(* CoDeSys 2.3.4.1 project: 20191210SRL乘3.pro *)
(* Libraries: Hollysys_PLC_COMM.lib 5.3.08 09:34:58, Hollysys_PLC_ANALOG.lib 28.12.05 14:28:34, Util.lib 28.10.11 18:19:34, SysLibVisu.lib 28.12.05 14:28:34, Hollysys_PLC_AnalogConvert.lib 5.3.08 09:47:22, Hollysys_PLC_Math.lib 7.3.06 16:53:32, Standard.lib 6.12.05 17:07:52, Hollysys_PLC_COMM2.lib 5.3.08 09:34:50, SYSLIBCALLBACK.LIB 6.12.05 17:07:52, Hollysys_PLC_Ex.lib 28.12.05 14:28:28, HS_PLC_ModebusMaster.lib 26.7.11 11:59:52 *)

(* PLC configuration (modules and I/O channels)
I AT %ID0 [DWORDInput_bit] 24 channels digital input
Q AT %QW0 [WordOutput3108_bit] 16 channels digital output(Relay)
LM3222 8×DO Relay [Ext_DO8_RELAY] node 0, in %IB4 out %QB2
  AT %QW2 [WordOutput_bit] 8 channels digital output(Relay)
LM3231 4×DI 4×DO Relay [Ext_DI4_DO4_RELAY] node 1, in %IB4 out %QB4
  AT %QW4 [WordOutput_bit] 4 channels digital output(Relay)
  AT %IW4 [WordInput_bit] 4 channels digital input
*)

(* POU PLC_PRG, LD *)
 PROGRAM PLC_PRG
VAR

	PSH_Q: BOOL;
	PSH_BL: BLINK;
	ET: TIME;
	KJ_SUO: BOOL;
	DY_SUO: BOOL;
	TD_TON: TON;
	TD_TON_Q: BOOL;
	PSH_BL_YSJ: BLINK;
	PSH_Q_YSJ: BOOL;
	JQ_1: JIQI_KONGZHI;
	JQ_2: JIQI_KONGZHI;
	JQ_JSH: ZJSHQ;
	CHD_1: BOOL;
	CHD_4: BOOL;
	CHD_3: BOOL;
	CHD_2: BOOL;
	BH_JQ_1: BAOHU_XIANSHI;
	YSJ_ONE_50_1: BOOL;
	YSJ_ONE_75_1: BOOL;
	YSJ_ONE_100_1: BOOL;
	YSJ_TWO_50_1: BOOL;
	YSJ_TWO_75_1: BOOL;
	YSJ_TWO_100_1: BOOL;
	T_DIAN: BOOL;
	T_R: R_TRIG;
	BH_JQ_2: BAOHU_XIANSHI;
	LN_SHB: BH_ZHFL;
	YOUFEN: YOU_FEN;

	MM_SUO: SUO;
	LN_FSH_1: BH_ZHFL;

	CHT: BOOL := 1;
	PW_OUT AT %MW892: INT;
	LN_FSH_2: BH_ZHFL;
	JT_KA: BOOL;
	YALI_OUT_1 AT %MW882: INT;
	PQ_YL_OUT AT %MW884: INT;
	PQ_XZH AT %MW364: INT;
	FAN_1_KA: BOOL;
	FAN_2_KA: BOOL;
	SHB_KA: BOOL;
	YL_KA: BOOL;
	PQYL: PQ_ZHFL_KZH;
	JZ_NJ_SHU_1: WORD;
	XUZH_IN_1 AT %MW476: INT;
	HIGH_IN_1 AT %MW478: INT;
	LOW_IN_1 AT %MW480: INT;
	XH_YSH_1: XH_YANSHI_1;
	XH_NJ_1: JQ_NJ_SHU;


	JJQ_DCF_1: BOOL;
	JQ_BJ_1: BJ_MIN_COOL;
	JQ_FUWEI_1: BJ_FUWEI;
	JQ_XHPX_1: XH_PAIXU;
	A_CX_1: BYTE;
	B_CX_1: BYTE;
       C_CX_1: BYTE;
	D_CX_1: BYTE;
	E_CX_1: BYTE;
	FU_WEI_1: BOOL;
	YSJ_ONE_1: BOOL;
	YSJ_TWO_1: BOOL;
	WBKZH: BOOL;
	XQ_1_T AT %MW886: INT;
	GRD_1_OUT AT %MW890: WORD;
	GRD_1_YSH: WORD;






	YL_FAN: BH_ZHFL;
	KF_ALA: BOOL;




	YSJ_CHD: BOOL;
	DY_JT: DY_JT_KZH;
	DY_JT_ALA: BOOL;
	CHD_5: BOOL;
	CHD_6: BOOL;
	F_CX_1: BYTE;
	YSJ_ONE: BOOL;
	YSJ_ONE_50: BOOL;
	YSJ_ONE_75: BOOL;
	YSJ_ONE_100: BOOL;
	YSJ_TWO: BOOL;
	YSJ_TWO_50: BOOL;
	YSJ_TWO_75: BOOL;
	YSJ_TWO_100: BOOL;
	YSJ_THREE: BOOL;
	YSJ_THREE_50: BOOL;
	YSJ_THREE_75: BOOL;
	YSJ_THREE_100: BOOL;
	YSJ_FOUR: BOOL;
	YSJ_FOUR_50: BOOL;
	YSJ_FOUR_75: BOOL;
	YSJ_FOUR_100: BOOL;
	YSJ_FIVE: BOOL;
	YSJ_FIVE_50: BOOL;
	YSJ_FIVE_75: BOOL;
	YSJ_FIVE_100: BOOL;
	YSJ_SIX: BOOL;
	YSJ_SIX_50: BOOL;
	YSJ_SIX_75: BOOL;
	YSJ_SIX_100: BOOL;

	BH_JQ_3: BAOHU_XIANSHI;
	JQ_3: JIQI_KONGZHI;
	BH_JQ_4: BAOHU_XIANSHI;
	JQ_4: JIQI_KONGZHI;
	BH_JQ_5: BAOHU_XIANSHI;
	JQ_5: JIQI_KONGZHI;
	BH_JQ_6: BAOHU_XIANSHI;
	JQ_6: JIQI_KONGZHI;
	PW_MN: MONI_LIANG_PW;

	PT_P: BLINK;

	GGD: AN_NIU;

	FAN_3_KA: BOOL;
	SHB2_KA: BOOL;
	FAN1: BH_ZHFL;
	FAN2: BH_ZHFL;
	FAN3: BH_ZHFL;
	YL: BH_ZHFL;
	SHB2: BH_ZHFL;
	SHB: BH_ZHFL;


	XQ_WD_XZH AT %MW470: INT;
	BH_WD AT %MW888: INT;
	PQ_YA_OUT AT %MW884: INT;


	Set_Local_Address: Set_Local_Address;
	MOUDBAS_OUT: BOOL;

	Analog_O: BOOL;
	FAN_4_KA: BOOL;
	OPEN_KJ: OPEN_KJ;
	FAN4: BH_ZHFL;






	R1_WD AT %MW1012: INT;
	R2_WD AT %MW1022: INT;
	R3_WD AT %MW1032: INT;
	R4_WD AT %MW1042: INT;
	R5_WD AT %MW1052: INT;
	R6_WD AT %MW1062: INT;
	R7_WD AT %MW1072: INT;
	R8_WD AT %MW1082: INT;

	R9_WD AT %MW1092: INT;
	R10_WD AT %MW1102: INT;
	R11_WD AT %MW1112: INT;
	R12_WD AT %MW1122: INT;
	R13_WD AT %MW1132: INT;
	R14_WD AT %MW1142: INT;






	K1: AN_NIU;
	K2: AN_NIU;
	K3: AN_NIU;
	K4: AN_NIU;
	K5: AN_NIU;
	K6: AN_NIU;
	K7: AN_NIU;
	K8: AN_NIU;
	K9: AN_NIU;
	K10: AN_NIU;
	K11: AN_NIU;
	K12: AN_NIU;
	K13: AN_NIU;
	K14: AN_NIU;


	K1_XZ AT %MW610: INT;
	K2_XZ AT %MW620: INT;
	K3_XZ AT %MW630: INT;
	K4_XZ AT %MW640: INT;
	K5_XZ AT %MW650: INT;
	K6_XZ AT %MW660: INT;
	K7_XZ AT %MW670: INT;
	K8_XZ AT %MW680: INT;
	K9_XZ AT %MW690: INT;
	K10_XZ AT %MW500: INT;
	K11_XZ AT %MW510: INT;
	K12_XZ AT %MW520: INT;
	K13_XZ AT %MW530: INT;
	K14_XZ AT %MW540: INT;

	K1_KJ AT %MW612: INT;
	K2_KJ AT %MW622: INT;
	K3_KJ AT %MW632: INT;
	K4_KJ AT %MW642: INT;
	K5_KJ AT %MW652: INT;
	K6_KJ AT %MW662: INT;
	K7_KJ AT %MW672: INT;
	K8_KJ AT %MW682: INT;
	K9_KJ AT %MW692: INT;
	K10_KJ AT %MW502: INT;
	K11_KJ AT %MW512: INT;
	K12_KJ AT %MW522: INT;
	K13_KJ AT %MW532: INT;
	K14_KJ AT %MW542: INT;


	K1_TJ AT %MW614: INT;
	K2_TJ AT %MW624: INT;
	K3_TJ AT %MW634: INT;
	K4_TJ AT %MW644: INT;
	K5_TJ AT %MW654: INT;
	K6_TJ AT %MW664: INT;
	K7_TJ AT %MW674: INT;
	K8_TJ AT %MW684: INT;
	K9_TJ AT %MW694: INT;
	K10_TJ AT %MW504: INT;
	K11_TJ AT %MW514: INT;
	K12_TJ AT %MW524: INT;
	K13_TJ AT %MW534: INT;
	K14_TJ AT %MW544: INT;

	K1_GS AT %MW616: INT;
	K2_GS AT %MW626: INT;
	K3_GS AT %MW636: INT;
	K4_GS AT %MW646: INT;
	K5_GS AT %MW656: INT;
	K6_GS AT %MW666: INT;
	K7_GS AT %MW676: INT;
	K8_GS AT %MW686: INT;
	K9_GS AT %MW696: INT;
	K10_GS AT %MW506: INT;
	K11_GS AT %MW516: INT;
	K12_GS AT %MW526: INT;
	K13_GS AT %MW536: INT;
	K14_GS AT %MW546: INT;


	DEF_1: BOOL;
	DEF_2: BOOL;
	DEF_3: BOOL;
	DEF_4: BOOL;
	DEF_5: BOOL;
	DEF_6: BOOL;
	DEF_7: BOOL;
	DEF_8: BOOL;
	DEF_9: BOOL;
	DEF_10: BOOL;
	DEF_11: BOOL;
	DEF_12: BOOL;
	DEF_13: BOOL;
	DEF_14: BOOL;
	DEF_1_DD: BOOL;
	DEF_2_DD: BOOL;
	DEF_3_DD: BOOL;
	DEF_4_DD: BOOL;
	DEF_5_DD: BOOL;
	DEF_6_DD: BOOL;
	DEF_7_DD: BOOL;
	DEF_8_DD: BOOL;
	DEF_9_DD: BOOL;
	DEF_10_DD: BOOL;
	DEF_11_DD: BOOL;
	DEF_12_DD: BOOL;
	DEF_13_DD: BOOL;
	DEF_14_DD: BOOL;
	ROOM1_ALA: BOOL;
	ROOM2_ALA: BOOL;
	ROOM3_ALA: BOOL;
	ROOM4_ALA: BOOL;
	ROOM5_ALA: BOOL;
	ROOM6_ALA: BOOL;
	ROOM7_ALA: BOOL;
	ROOM8_ALA: BOOL;
	ROOM9_ALA: BOOL;
	ROOM10_ALA: BOOL;
	ROOM11_ALA: BOOL;
	ROOM12_ALA: BOOL;
	ROOM13_ALA: BOOL;
	ROOM14_ALA: BOOL;
	COOL_1_M: DWORD;
	COOL_2_M: DWORD;
	COOL_3_M: DWORD;
	COOL_4_M: DWORD;
	COOL_5_M: DWORD;
	COOL_6_M: DWORD;
	COOL_7_M: DWORD;
	COOL_8_M: DWORD;
	COOL_9_M: DWORD;
	COOL_10_M: DWORD;
	COOL_11_M: DWORD;
	COOL_12_M: DWORD;
	COOL_13_M: DWORD;
	COOL_14_M: DWORD;
	ROOM1_T_ZT: WORD;
	ROOM2_T_ZT: WORD;
	ROOM3_T_ZT: WORD;
	ROOM4_T_ZT: WORD;
	ROOM5_T_ZT: WORD;
	ROOM6_T_ZT: WORD;
	ROOM7_T_ZT: WORD;
	ROOM8_T_ZT: WORD;
	ROOM9_T_ZT: WORD;
	ROOM10_T_ZT: WORD;
	ROOM11_T_ZT: WORD;
	ROOM12_T_ZT: WORD;
	ROOM13_T_ZT: WORD;
	ROOM14_T_ZT: WORD;
	BZH_1_M: DWORD;
	BZH_2_M: DWORD;
	BZH_3_M: DWORD;
	BZH_4_M: DWORD;
	BZH_5_M: DWORD;
	BZH_6_M: DWORD;
	BZH_7_M: DWORD;
	BZH_8_M: DWORD;
	BZH_9_M: DWORD;
	BZH_10_M: DWORD;
	BZH_11_M: DWORD;
	BZH_12_M: DWORD;
	BZH_13_M: DWORD;
	BZH_14_M: DWORD;

	DEF_1_ZD: BOOL;
	DEF_2_ZD: BOOL;
	DEF_3_ZD: BOOL;
	DEF_4_ZD: BOOL;
	DEF_5_ZD: BOOL;
	DEF_6_ZD: BOOL;
	DEF_7_ZD: BOOL;
	DEF_8_ZD: BOOL;
	DEF_9_ZD: BOOL;
	DEF_10_ZD: BOOL;
	DEF_11_ZD: BOOL;
	DEF_12_ZD: BOOL;
	DEF_13_ZD: BOOL;
	DEF_14_ZD: BOOL;

	DEF_1_FJ: BOOL;
	DEF_2_FJ: BOOL;
	DEF_3_FJ: BOOL;
	DEF_4_FJ: BOOL;
	DEF_5_FJ: BOOL;
	DEF_6_FJ: BOOL;
	DEF_7_FJ: BOOL;
	DEF_8_FJ: BOOL;
	DEF_9_FJ: BOOL;
	DEF_10_FJ: BOOL;
	DEF_11_FJ: BOOL;
	DEF_12_FJ: BOOL;
	DEF_13_FJ: BOOL;
	DEF_14_FJ: BOOL;

	ROOM_1_FJ: BOOL;
	ROOM_2_FJ: BOOL;
	ROOM_3_FJ: BOOL;
	ROOM_4_FJ: BOOL;
	ROOM_5_FJ: BOOL;
	ROOM_6_FJ: BOOL;
	ROOM_7_FJ: BOOL;
	ROOM_8_FJ: BOOL;
	ROOM_9_FJ: BOOL;
	ROOM_10_FJ: BOOL;
	ROOM_11_FJ: BOOL;
	ROOM_12_FJ: BOOL;
	ROOM_13_FJ: BOOL;
	ROOM_14_FJ: BOOL;



	DEF_YUNSUAN: DEF_YUNSUAN;

	CS_SHB: BH_ZHFL;
	YL_K: BH_ZHFL;

	CF: BLINK;

	Analog_: BOOL;
	OPEN_K: OPEN_KJ;
	Analog_IN1: Analog_IN;
	Analog_OUT1: BOOL;
	Analog_IN2: Analog_IN;
	Analog_OUT2: BOOL;

	FB1_CHD: BOOL;
	FB1_ALA: BOOL;
	FB2_CHD: BOOL;
	FB2_ALA: BOOL;

	FB_AN: AN_NIU;
	FB_TON: TON;
	YW_XSH AT %MW1200: INT;
	SS: BOOL;


	B1: BOOL;
	B3: BOOL;
	B2: BOOL;
	XZ_NIU: AN_NIU;
	BY_NIU: AN_NIU;
	FB_CHD: BOOL;
	WBKZH1: BOOL;
	PQ_GRD: PQ_GRD;
	PQ_BH_WD AT %MW906: INT;
	PQ_GRD_OUT AT %MW908: INT;
	PQ_GRD_SET AT %MW490: INT;
	HQ_WD_XZ AT %MW598: INT;
	KCHD_1: BOOL;
	KCHD_2: BOOL;
	KCHD_3: BOOL;
	KCHD_4: BOOL;
	DEF_SHB: BH_ZHFL;

	Analog_IN3: Analog_IN;
	Analog_OUT3: BOOL;

	TT_BH_WCH AT %MW448: INT;
	SHB_YAN: YANSHI_CLOSE;
	SHL_YSH_SET AT %MW468: WORD;
	SHL_YSH_SET_0: BOOL;
	SHL_T: YANSHI_OPEN;
	SHL_BH: SHL_BH;
	KJ: BOOL;
	SHB1: BOOL;

	T1 AT %MW1300: INT;
	T2 AT %MW1302: INT;
	JQ_BJ: BJ_MIN_COOL_1;
	JQ_FUWEI: BJ_FUWEI_1;
	FW_1: BOOL;
	FW_3: BOOL;
	FW_2: BOOL;
	FW_4: BOOL;
	FW_5: BOOL;
	FW_6: BOOL;
	CX_1: BYTE;
	CX_2: BYTE;
	CX_3: BYTE;
	CX_4: BYTE;
	CX_5: BYTE;
	CX_6: BYTE;




	WD_XH1: WD_XH;
	K1_IN: INT;
	K1_T1 AT %MW1300: INT;
	K1_T2 AT %MW1302: INT;
	K1_T3 AT %MW1304: INT;
	K1_T4 AT %MW1306: INT;

	K2_T1 AT %MW1308: INT;
	K2_T2 AT %MW1310: INT;
	K2_T3 AT %MW1312: INT;
	K2_T4 AT %MW1314: INT;

	K3_T1 AT %MW1316: INT;
	K3_T2 AT %MW1318: INT;

	K3_T4 AT %MW1322: INT;
	K4_T1 AT %MW1324: INT;
	K4_T2 AT %MW1326: INT;
	K4_T3 AT %MW1328: INT;
	K4_T4 AT %MW1330: INT;

	K2_IN: INT;
	WD_XH2: WD_XH;
	WD_XH3: WD_XH;
	K3_IN: INT;
	WD_XH4: WD_XH;
	K4_IN: INT;

	K3_T3 AT %MW1320: INT;
	Reset_COMM2_PRMT: Reset_COMM2_PRMT;
	Reset_COMM2_: BOOL;
	BLINK: BLINK;
	ModbusMaster485: ModbusMaster485;
	DDD: BYTE;
	ModbusMaster: BOOL;
	H: BOOL;
	O: BOOL;
	KCHD_5: BOOL;
	JQ_SHU: WORD;
	YL_DCF2: BOOL;
	TON_GYW: TON;
	SHB_AN: AN_NIU;
	BLINK_SHB: BLINK;
	SHB_XHKA: BOOL;
	YF_WD AT %MW1332: INT;
	K_1: BOOL;
	K_2: BOOL;
	YA_ALA: BOOL;
	YA AT %MW1332: INT;
	YA_CHA AT %MW1334: INT;
	SET_YA AT %MW618: INT;
	Y_K: BOOL;
	JJQ: BOOL;
	JJQ_K AT %MW628: INT;
	JJQ_G AT %MW638: INT;
	BB: BB;
	HIGH_IN_2 AT %MW648: INT;
	LOW_IN_2 AT %MW658: INT;
END_VAR
VAR RETAIN

END_VAR
VAR RETAIN
END_VAR
VAR_INPUT
END_VAR
VAR_OUTPUT
END_VAR
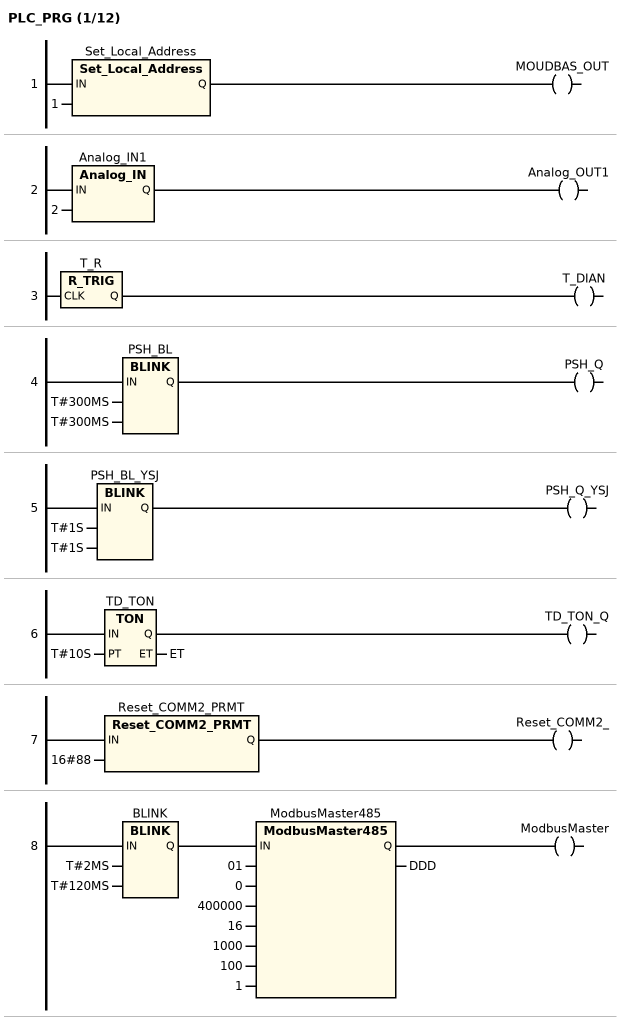
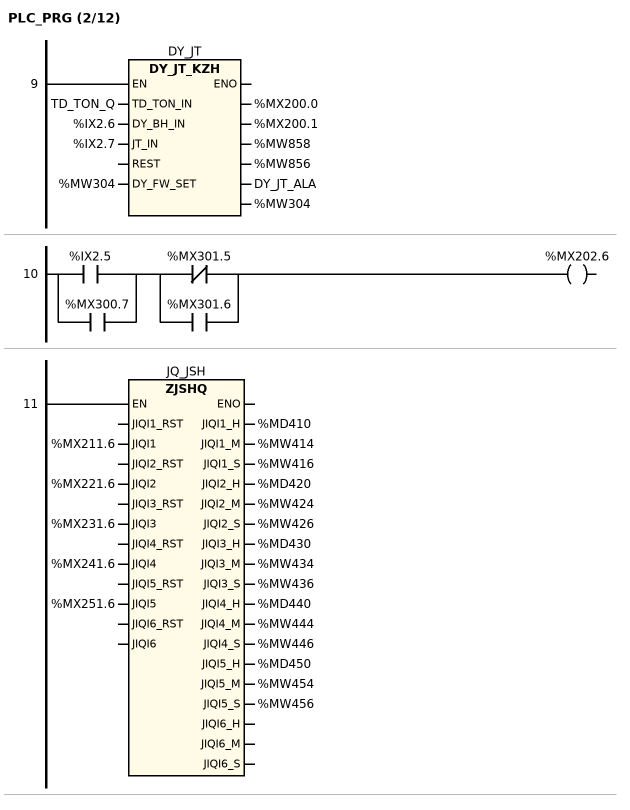
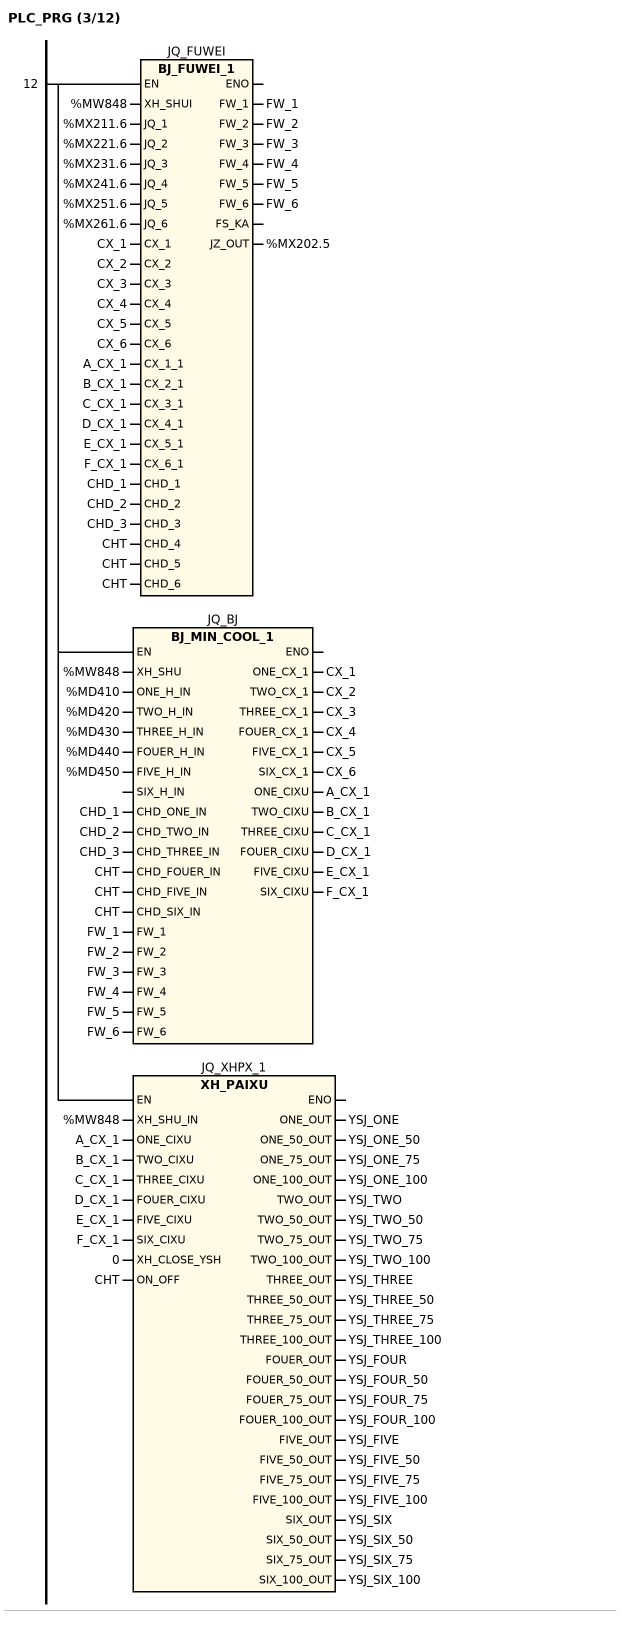
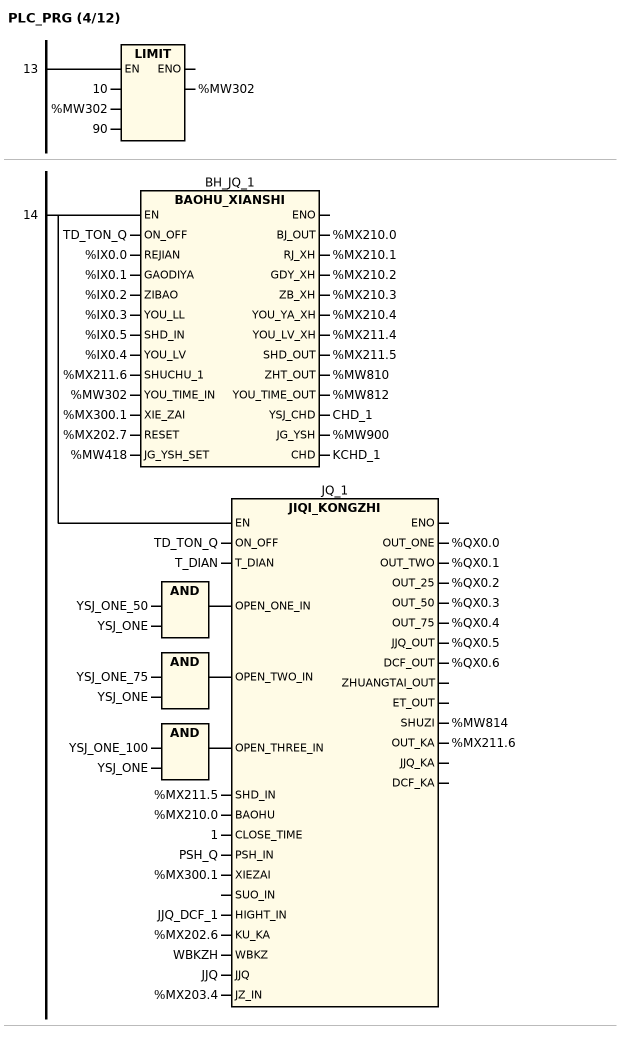
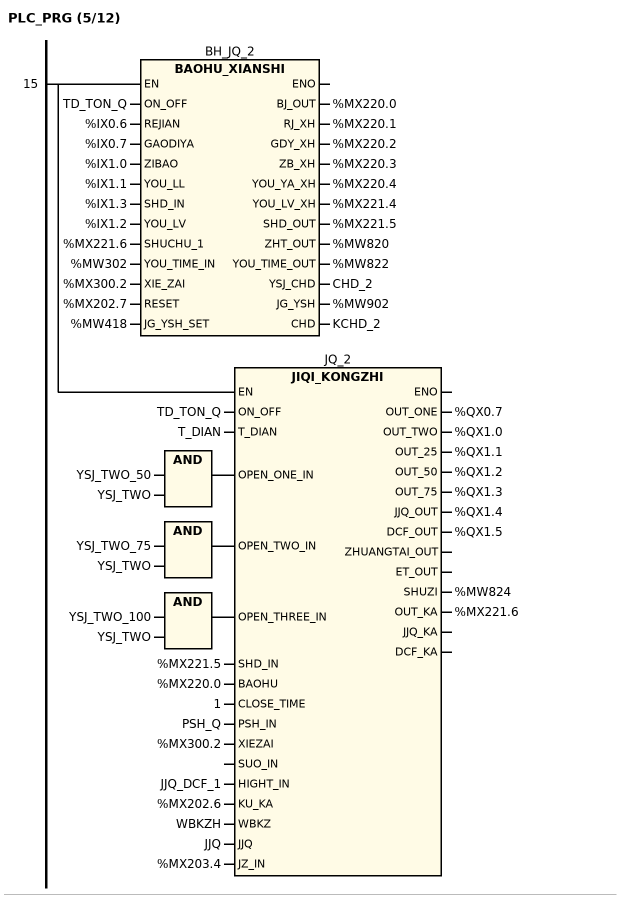
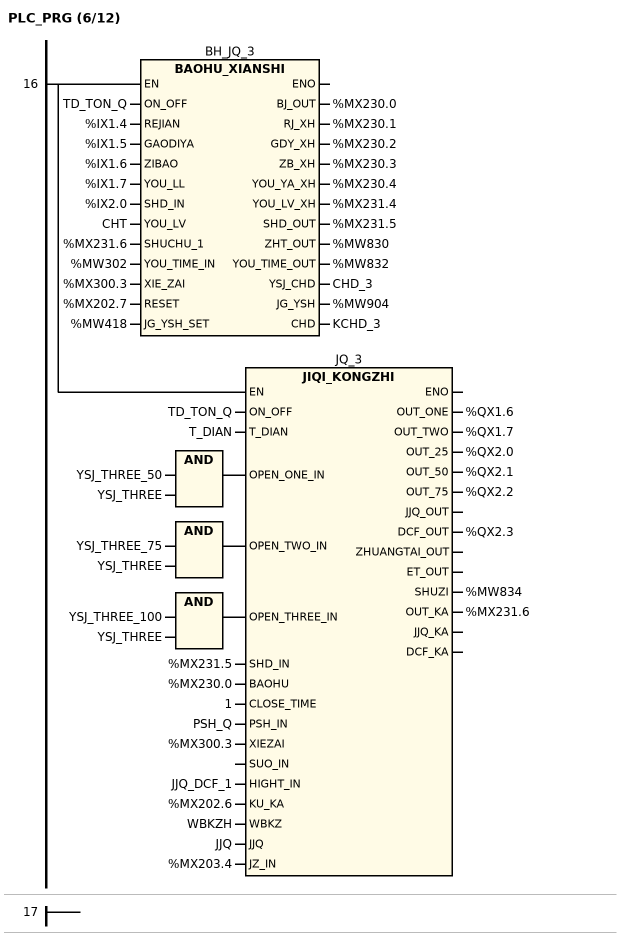
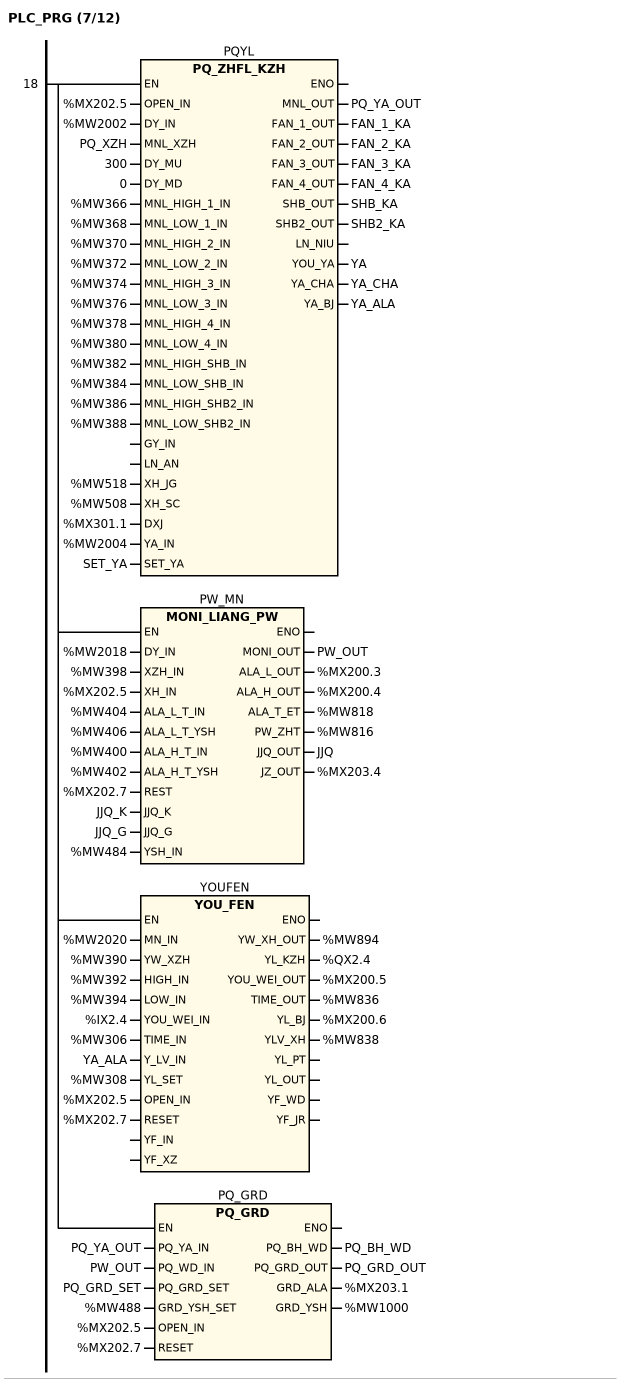
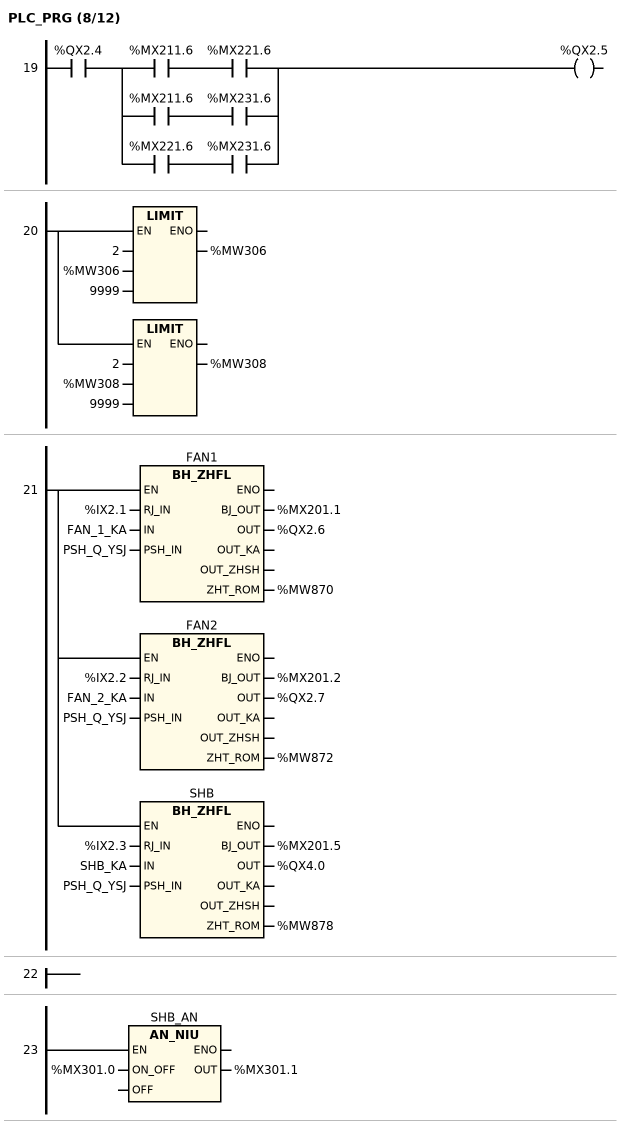
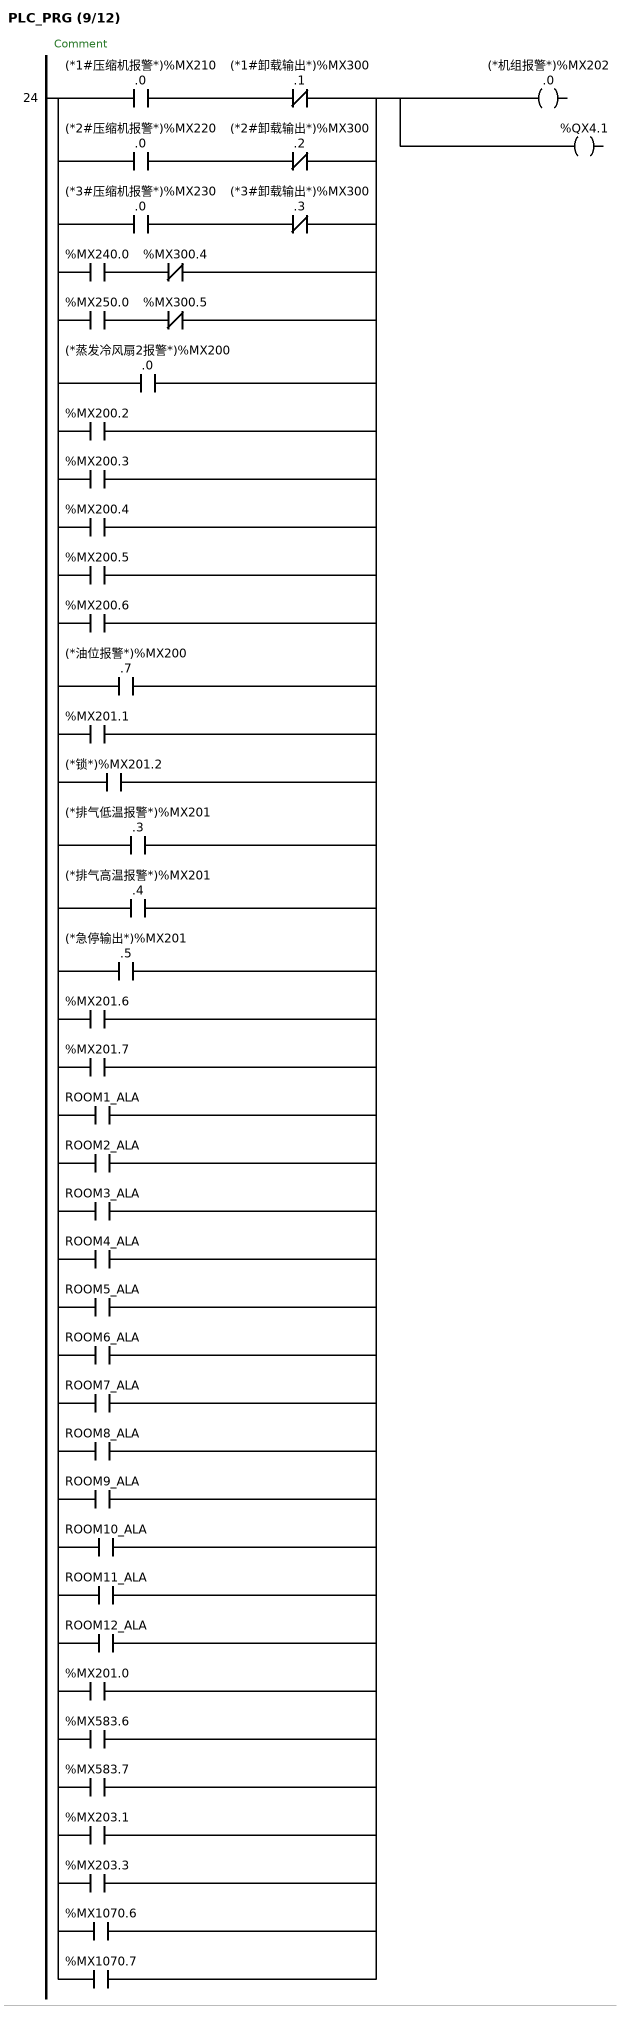
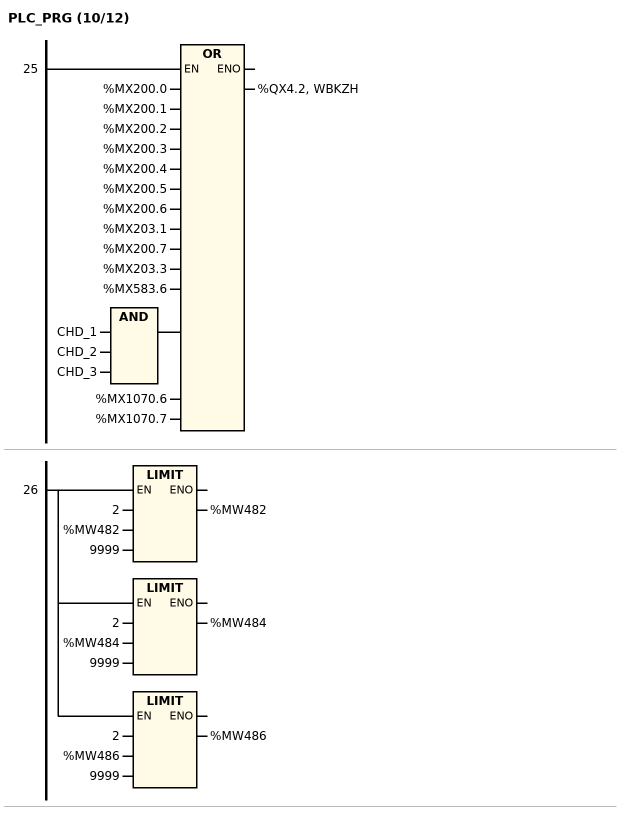
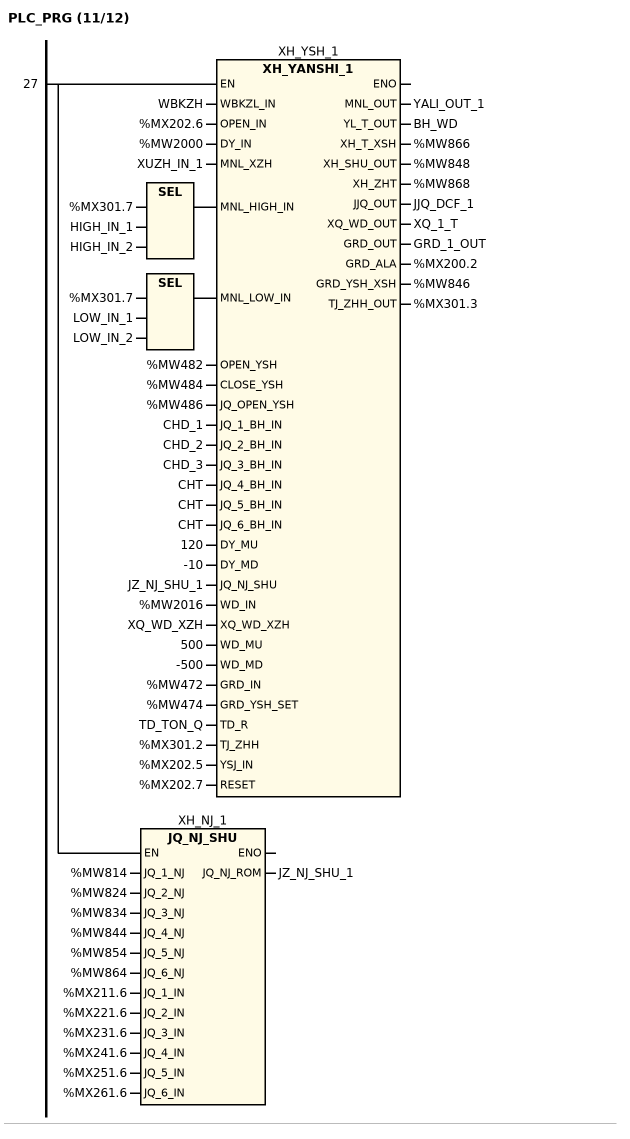
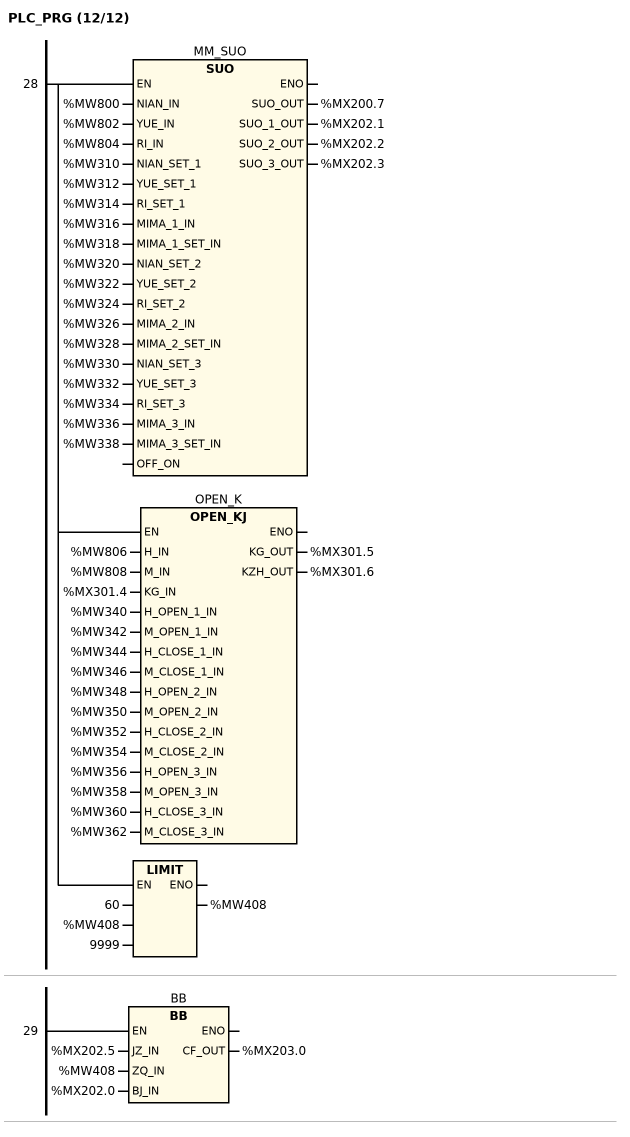
_LD_ (* Ladder Diagram *)
NETWORK 1
	Set_Local_Address:Set_Local_Address(*, 1) --- (MOUDBAS_OUT)
NETWORK 2
	Analog_IN1:Analog_IN(*, 2) --- (Analog_OUT1)
NETWORK 3
	T_R:R_TRIG(CLK: *) --- (T_DIAN)
NETWORK 4
	PSH_BL:BLINK(*, T#300MS, T#300MS) --- (PSH_Q)
NETWORK 5
	PSH_BL_YSJ:BLINK(*, T#1S, T#1S) --- (PSH_Q_YSJ)
NETWORK 6
	TD_TON:TON(IN: *, PT: T#10S, ET => ET) --- (TD_TON_Q)
NETWORK 7
	Reset_COMM2_PRMT:Reset_COMM2_PRMT(*, 16#88) --- (Reset_COMM2_)
NETWORK 8
	BLINK:BLINK(*, T#2MS, T#120MS) - ModbusMaster485:ModbusMaster485(*, 01, 0, 400000, 16, 1000, 100, 1, out 2 => DDD) --- (ModbusMaster)
NETWORK 9
	*
		EN --- DY_JT:DY_JT_KZH(TD_TON_IN: TD_TON_Q, DY_BH_IN: %IX2.6, JT_IN: %IX2.7, REST: , DY_FW_SET: %MW304, out 2 => %MX200.1, out 3 => %MW858, out 4 => %MW856, out 5 => DY_JT_ALA, out 6 => %MW304) => %MX200.0
NETWORK 10
	{ [%IX2.5] | [%MX300.7] } - { [/%MX301.5] | [%MX301.6] } --- (%MX202.6)
NETWORK 11
	*
		EN --- JQ_JSH:ZJSHQ(JIQI1_RST: , JIQI1: %MX211.6, JIQI2_RST: , JIQI2: %MX221.6, JIQI3_RST: , JIQI3: %MX231.6, JIQI4_RST: , JIQI4: %MX241.6, JIQI5_RST: , JIQI5: %MX251.6, JIQI6_RST: , JIQI6: , JIQI1_M => %MW414, JIQI1_S => %MW416, JIQI2_H => %MD420, JIQI2_M => %MW424, JIQI2_S => %MW426, JIQI3_H => %MD430, JIQI3_M => %MW434, JIQI3_S => %MW436, JIQI4_H => %MD440, JIQI4_M => %MW444, JIQI4_S => %MW446, JIQI5_H => %MD450, JIQI5_M => %MW454, JIQI5_S => %MW456) => %MD410
NETWORK 12
	*
		EN --- JQ_FUWEI:BJ_FUWEI_1(XH_SHUI: %MW848, JQ_1: %MX211.6, JQ_2: %MX221.6, JQ_3: %MX231.6, JQ_4: %MX241.6, JQ_5: %MX251.6, JQ_6: %MX261.6, CX_1: CX_1, CX_2: CX_2, CX_3: CX_3, CX_4: CX_4, CX_5: CX_5, CX_6: CX_6, CX_1_1: A_CX_1, CX_2_1: B_CX_1, CX_3_1: C_CX_1, CX_4_1: D_CX_1, CX_5_1: E_CX_1, CX_6_1: F_CX_1, CHD_1: CHD_1, CHD_2: CHD_2, CHD_3: CHD_3, CHD_4: CHT, CHD_5: CHT, CHD_6: CHT, FW_2 => FW_2, FW_3 => FW_3, FW_4 => FW_4, FW_5 => FW_5, FW_6 => FW_6, JZ_OUT => %MX202.5) => FW_1
		EN --- JQ_BJ:BJ_MIN_COOL_1(XH_SHU: %MW848, ONE_H_IN: %MD410, TWO_H_IN: %MD420, THREE_H_IN: %MD430, FOUER_H_IN: %MD440, FIVE_H_IN: %MD450, SIX_H_IN: , CHD_ONE_IN: CHD_1, CHD_TWO_IN: CHD_2, CHD_THREE_IN: CHD_3, CHD_FOUER_IN: CHT, CHD_FIVE_IN: CHT, CHD_SIX_IN: CHT, FW_1: FW_1, FW_2: FW_2, FW_3: FW_3, FW_4: FW_4, FW_5: FW_5, FW_6: FW_6, TWO_CX_1 => CX_2, THREE_CX_1 => CX_3, FOUER_CX_1 => CX_4, FIVE_CX_1 => CX_5, SIX_CX_1 => CX_6, ONE_CIXU => A_CX_1, TWO_CIXU => B_CX_1, THREE_CIXU => C_CX_1, FOUER_CIXU => D_CX_1, FIVE_CIXU => E_CX_1, SIX_CIXU => F_CX_1) => CX_1
		EN --- JQ_XHPX_1:XH_PAIXU(XH_SHU_IN: %MW848, ONE_CIXU: A_CX_1, TWO_CIXU: B_CX_1, THREE_CIXU: C_CX_1, FOUER_CIXU: D_CX_1, FIVE_CIXU: E_CX_1, SIX_CIXU: F_CX_1, XH_CLOSE_YSH: 0, ON_OFF: CHT, ONE_50_OUT => YSJ_ONE_50, ONE_75_OUT => YSJ_ONE_75, ONE_100_OUT => YSJ_ONE_100, TWO_OUT => YSJ_TWO, TWO_50_OUT => YSJ_TWO_50, TWO_75_OUT => YSJ_TWO_75, TWO_100_OUT => YSJ_TWO_100, THREE_OUT => YSJ_THREE, THREE_50_OUT => YSJ_THREE_50, THREE_75_OUT => YSJ_THREE_75, THREE_100_OUT => YSJ_THREE_100, FOUER_OUT => YSJ_FOUR, FOUER_50_OUT => YSJ_FOUR_50, FOUER_75_OUT => YSJ_FOUR_75, FOUER_100_OUT => YSJ_FOUR_100, FIVE_OUT => YSJ_FIVE, FIVE_50_OUT => YSJ_FIVE_50, FIVE_75_OUT => YSJ_FIVE_75, FIVE_100_OUT => YSJ_FIVE_100, SIX_OUT => YSJ_SIX, SIX_50_OUT => YSJ_SIX_50, SIX_75_OUT => YSJ_SIX_75, SIX_100_OUT => YSJ_SIX_100) => YSJ_ONE
NETWORK 13
	*
		EN --- LIMIT(10, %MW302, 90) => %MW302
NETWORK 14
	*
		EN --- BH_JQ_1:BAOHU_XIANSHI(ON_OFF: TD_TON_Q, REJIAN: %IX0.0, GAODIYA: %IX0.1, ZIBAO: %IX0.2, YOU_LL: %IX0.3, SHD_IN: %IX0.5, YOU_LV: %IX0.4, SHUCHU_1: %MX211.6, YOU_TIME_IN: %MW302, XIE_ZAI: %MX300.1, RESET: %MX202.7, JG_YSH_SET: %MW418, RJ_XH => %MX210.1, GDY_XH => %MX210.2, ZB_XH => %MX210.3, YOU_YA_XH => %MX210.4, YOU_LV_XH => %MX211.4, SHD_OUT => %MX211.5, ZHT_OUT => %MW810, YOU_TIME_OUT => %MW812, YSJ_CHD => CHD_1, JG_YSH => %MW900, CHD => KCHD_1) => %MX210.0
		EN --- JQ_1:JIQI_KONGZHI(ON_OFF: TD_TON_Q, T_DIAN: T_DIAN, OPEN_ONE_IN: AND(YSJ_ONE_50, YSJ_ONE), OPEN_TWO_IN: AND(YSJ_ONE_75, YSJ_ONE), OPEN_THREE_IN: AND(YSJ_ONE_100, YSJ_ONE), SHD_IN: %MX211.5, BAOHU: %MX210.0, CLOSE_TIME: 1, PSH_IN: PSH_Q, XIEZAI: %MX300.1, SUO_IN: , HIGHT_IN: JJQ_DCF_1, KU_KA: %MX202.6, WBKZ: WBKZH, JJQ: JJQ, JZ_IN: %MX203.4, OUT_TWO => %QX0.1, OUT_25 => %QX0.2, OUT_50 => %QX0.3, OUT_75 => %QX0.4, JJQ_OUT => %QX0.5, DCF_OUT => %QX0.6, SHUZI => %MW814, OUT_KA => %MX211.6) => %QX0.0
NETWORK 15
	*
		EN --- BH_JQ_2:BAOHU_XIANSHI(ON_OFF: TD_TON_Q, REJIAN: %IX0.6, GAODIYA: %IX0.7, ZIBAO: %IX1.0, YOU_LL: %IX1.1, SHD_IN: %IX1.3, YOU_LV: %IX1.2, SHUCHU_1: %MX221.6, YOU_TIME_IN: %MW302, XIE_ZAI: %MX300.2, RESET: %MX202.7, JG_YSH_SET: %MW418, RJ_XH => %MX220.1, GDY_XH => %MX220.2, ZB_XH => %MX220.3, YOU_YA_XH => %MX220.4, YOU_LV_XH => %MX221.4, SHD_OUT => %MX221.5, ZHT_OUT => %MW820, YOU_TIME_OUT => %MW822, YSJ_CHD => CHD_2, JG_YSH => %MW902, CHD => KCHD_2) => %MX220.0
		EN --- JQ_2:JIQI_KONGZHI(ON_OFF: TD_TON_Q, T_DIAN: T_DIAN, OPEN_ONE_IN: AND(YSJ_TWO_50, YSJ_TWO), OPEN_TWO_IN: AND(YSJ_TWO_75, YSJ_TWO), OPEN_THREE_IN: AND(YSJ_TWO_100, YSJ_TWO), SHD_IN: %MX221.5, BAOHU: %MX220.0, CLOSE_TIME: 1, PSH_IN: PSH_Q, XIEZAI: %MX300.2, SUO_IN: , HIGHT_IN: JJQ_DCF_1, KU_KA: %MX202.6, WBKZ: WBKZH, JJQ: JJQ, JZ_IN: %MX203.4, OUT_TWO => %QX1.0, OUT_25 => %QX1.1, OUT_50 => %QX1.2, OUT_75 => %QX1.3, JJQ_OUT => %QX1.4, DCF_OUT => %QX1.5, SHUZI => %MW824, OUT_KA => %MX221.6) => %QX0.7
NETWORK 16
	*
		EN --- BH_JQ_3:BAOHU_XIANSHI(ON_OFF: TD_TON_Q, REJIAN: %IX1.4, GAODIYA: %IX1.5, ZIBAO: %IX1.6, YOU_LL: %IX1.7, SHD_IN: %IX2.0, YOU_LV: CHT, SHUCHU_1: %MX231.6, YOU_TIME_IN: %MW302, XIE_ZAI: %MX300.3, RESET: %MX202.7, JG_YSH_SET: %MW418, RJ_XH => %MX230.1, GDY_XH => %MX230.2, ZB_XH => %MX230.3, YOU_YA_XH => %MX230.4, YOU_LV_XH => %MX231.4, SHD_OUT => %MX231.5, ZHT_OUT => %MW830, YOU_TIME_OUT => %MW832, YSJ_CHD => CHD_3, JG_YSH => %MW904, CHD => KCHD_3) => %MX230.0
		EN --- JQ_3:JIQI_KONGZHI(ON_OFF: TD_TON_Q, T_DIAN: T_DIAN, OPEN_ONE_IN: AND(YSJ_THREE_50, YSJ_THREE), OPEN_TWO_IN: AND(YSJ_THREE_75, YSJ_THREE), OPEN_THREE_IN: AND(YSJ_THREE_100, YSJ_THREE), SHD_IN: %MX231.5, BAOHU: %MX230.0, CLOSE_TIME: 1, PSH_IN: PSH_Q, XIEZAI: %MX300.3, SUO_IN: , HIGHT_IN: JJQ_DCF_1, KU_KA: %MX202.6, WBKZ: WBKZH, JJQ: JJQ, JZ_IN: %MX203.4, OUT_TWO => %QX1.7, OUT_25 => %QX2.0, OUT_50 => %QX2.1, OUT_75 => %QX2.2, DCF_OUT => %QX2.3, SHUZI => %MW834, OUT_KA => %MX231.6) => %QX1.6
NETWORK 17
	*
NETWORK 18
	*
		EN --- PQYL:PQ_ZHFL_KZH(OPEN_IN: %MX202.5, DY_IN: %MW2002, MNL_XZH: PQ_XZH, DY_MU: 300, DY_MD: 0, MNL_HIGH_1_IN: %MW366, MNL_LOW_1_IN: %MW368, MNL_HIGH_2_IN: %MW370, MNL_LOW_2_IN: %MW372, MNL_HIGH_3_IN: %MW374, MNL_LOW_3_IN: %MW376, MNL_HIGH_4_IN: %MW378, MNL_LOW_4_IN: %MW380, MNL_HIGH_SHB_IN: %MW382, MNL_LOW_SHB_IN: %MW384, MNL_HIGH_SHB2_IN: %MW386, MNL_LOW_SHB2_IN: %MW388, GY_IN: , LN_AN: , XH_JG: %MW518, XH_SC: %MW508, DXJ: %MX301.1, YA_IN: %MW2004, SET_YA: SET_YA, FAN_1_OUT => FAN_1_KA, FAN_2_OUT => FAN_2_KA, FAN_3_OUT => FAN_3_KA, FAN_4_OUT => FAN_4_KA, SHB_OUT => SHB_KA, SHB2_OUT => SHB2_KA, YOU_YA => YA, YA_CHA => YA_CHA, YA_BJ => YA_ALA) => PQ_YA_OUT
		EN --- PW_MN:MONI_LIANG_PW(DY_IN: %MW2018, XZH_IN: %MW398, XH_IN: %MX202.5, ALA_L_T_IN: %MW404, ALA_L_T_YSH: %MW406, ALA_H_T_IN: %MW400, ALA_H_T_YSH: %MW402, REST: %MX202.7, JJQ_K: JJQ_K, JJQ_G: JJQ_G, YSH_IN: %MW484, ALA_L_OUT => %MX200.3, ALA_H_OUT => %MX200.4, ALA_T_ET => %MW818, PW_ZHT => %MW816, JJQ_OUT => JJQ, JZ_OUT => %MX203.4) => PW_OUT
		EN --- YOUFEN:YOU_FEN(MN_IN: %MW2020, YW_XZH: %MW390, HIGH_IN: %MW392, LOW_IN: %MW394, YOU_WEI_IN: %IX2.4, TIME_IN: %MW306, Y_LV_IN: YA_ALA, YL_SET: %MW308, OPEN_IN: %MX202.5, RESET: %MX202.7, YF_IN: , YF_XZ: , YL_KZH => %QX2.4, YOU_WEI_OUT => %MX200.5, TIME_OUT => %MW836, YL_BJ => %MX200.6, YLV_XH => %MW838) => %MW894
		EN --- PQ_GRD:PQ_GRD(PQ_YA_IN: PQ_YA_OUT, PQ_WD_IN: PW_OUT, PQ_GRD_SET: PQ_GRD_SET, GRD_YSH_SET: %MW488, OPEN_IN: %MX202.5, RESET: %MX202.7, PQ_GRD_OUT => PQ_GRD_OUT, GRD_ALA => %MX203.1, GRD_YSH => %MW1000) => PQ_BH_WD
NETWORK 19
	[%QX2.4] - { [%MX211.6] - [%MX221.6] | [%MX211.6] - [%MX231.6] | [%MX221.6] - [%MX231.6] } --- (%QX2.5)
NETWORK 20
	*
		EN --- LIMIT(2, %MW306, 9999) => %MW306
		EN --- LIMIT(2, %MW308, 9999) => %MW308
NETWORK 21
	*
		EN --- FAN1:BH_ZHFL(RJ_IN: %IX2.1, IN: FAN_1_KA, PSH_IN: PSH_Q_YSJ, OUT => %QX2.6, ZHT_ROM => %MW870) => %MX201.1
		EN --- FAN2:BH_ZHFL(RJ_IN: %IX2.2, IN: FAN_2_KA, PSH_IN: PSH_Q_YSJ, OUT => %QX2.7, ZHT_ROM => %MW872) => %MX201.2
		EN --- SHB:BH_ZHFL(RJ_IN: %IX2.3, IN: SHB_KA, PSH_IN: PSH_Q_YSJ, OUT => %QX4.0, ZHT_ROM => %MW878) => %MX201.5
NETWORK 22
	*
NETWORK 23
	*
		EN --- SHB_AN:AN_NIU(ON_OFF: %MX301.0, OFF: ) => %MX301.1
NETWORK 24 (* Comment *)
	{ [(*1#压缩机报警*)%MX210.0] - [/(*1#卸载输出*)%MX300.1] | [(*2#压缩机报警*)%MX220.0] - [/(*2#卸载输出*)%MX300.2] | [(*3#压缩机报警*)%MX230.0] - [/(*3#卸载输出*)%MX300.3] | [%MX240.0] - [/%MX300.4] | [%MX250.0] - [/%MX300.5] | [(*蒸发冷风扇2报警*)%MX200.0] | [%MX200.2] | [%MX200.3] | [%MX200.4] | [%MX200.5] | [%MX200.6] | [(*油位报警*)%MX200.7] | [%MX201.1] | [(*锁*)%MX201.2] | [(*排气低温报警*)%MX201.3] | [(*排气高温报警*)%MX201.4] | [(*急停输出*)%MX201.5] | [%MX201.6] | [%MX201.7] | [ROOM1_ALA] | [ROOM2_ALA] | [ROOM3_ALA] | [ROOM4_ALA] | [ROOM5_ALA] | [ROOM6_ALA] | [ROOM7_ALA] | [ROOM8_ALA] | [ROOM9_ALA] | [ROOM10_ALA] | [ROOM11_ALA] | [ROOM12_ALA] | [%MX201.0] | [%MX583.6] | [%MX583.7] | [%MX203.1] | [%MX203.3] | [%MX1070.6] | [%MX1070.7] } --- ((*机组报警*)%MX202.0) (%QX4.1)
NETWORK 25
	*
		EN --- OR(%MX200.0, %MX200.1, %MX200.2, %MX200.3, %MX200.4, %MX200.5, %MX200.6, %MX203.1, %MX200.7, %MX203.3, %MX583.6, AND(CHD_1, CHD_2, CHD_3), %MX1070.6, %MX1070.7) => %QX4.2, WBKZH
NETWORK 26
	*
		EN --- LIMIT(2, %MW482, 9999) => %MW482
		EN --- LIMIT(2, %MW484, 9999) => %MW484
		EN --- LIMIT(2, %MW486, 9999) => %MW486
NETWORK 27
	*
		EN --- XH_YSH_1:XH_YANSHI_1(WBKZL_IN: WBKZH, OPEN_IN: %MX202.6, DY_IN: %MW2000, MNL_XZH: XUZH_IN_1, MNL_HIGH_IN: SEL(%MX301.7, HIGH_IN_1, HIGH_IN_2), MNL_LOW_IN: SEL(%MX301.7, LOW_IN_1, LOW_IN_2), OPEN_YSH: %MW482, CLOSE_YSH: %MW484, JQ_OPEN_YSH: %MW486, JQ_1_BH_IN: CHD_1, JQ_2_BH_IN: CHD_2, JQ_3_BH_IN: CHD_3, JQ_4_BH_IN: CHT, JQ_5_BH_IN: CHT, JQ_6_BH_IN: CHT, DY_MU: 120, DY_MD: -10, JQ_NJ_SHU: JZ_NJ_SHU_1, WD_IN: %MW2016, XQ_WD_XZH: XQ_WD_XZH, WD_MU: 500, WD_MD: -500, GRD_IN: %MW472, GRD_YSH_SET: %MW474, TD_R: TD_TON_Q, TJ_ZHH: %MX301.2, YSJ_IN: %MX202.5, RESET: %MX202.7, YL_T_OUT => BH_WD, XH_T_XSH => %MW866, XH_SHU_OUT => %MW848, XH_ZHT => %MW868, JJQ_OUT => JJQ_DCF_1, XQ_WD_OUT => XQ_1_T, GRD_OUT => GRD_1_OUT, GRD_ALA => %MX200.2, GRD_YSH_XSH => %MW846, TJ_ZHH_OUT => %MX301.3) => YALI_OUT_1
		EN --- XH_NJ_1:JQ_NJ_SHU(JQ_1_NJ: %MW814, JQ_2_NJ: %MW824, JQ_3_NJ: %MW834, JQ_4_NJ: %MW844, JQ_5_NJ: %MW854, JQ_6_NJ: %MW864, JQ_1_IN: %MX211.6, JQ_2_IN: %MX221.6, JQ_3_IN: %MX231.6, JQ_4_IN: %MX241.6, JQ_5_IN: %MX251.6, JQ_6_IN: %MX261.6) => JZ_NJ_SHU_1
NETWORK 28
	*
		EN --- MM_SUO:SUO(NIAN_IN: %MW800, YUE_IN: %MW802, RI_IN: %MW804, NIAN_SET_1: %MW310, YUE_SET_1: %MW312, RI_SET_1: %MW314, MIMA_1_IN: %MW316, MIMA_1_SET_IN: %MW318, NIAN_SET_2: %MW320, YUE_SET_2: %MW322, RI_SET_2: %MW324, MIMA_2_IN: %MW326, MIMA_2_SET_IN: %MW328, NIAN_SET_3: %MW330, YUE_SET_3: %MW332, RI_SET_3: %MW334, MIMA_3_IN: %MW336, MIMA_3_SET_IN: %MW338, OFF_ON: , SUO_1_OUT => %MX202.1, SUO_2_OUT => %MX202.2, SUO_3_OUT => %MX202.3) => %MX200.7
		EN --- OPEN_K:OPEN_KJ(H_IN: %MW806, M_IN: %MW808, KG_IN: %MX301.4, H_OPEN_1_IN: %MW340, M_OPEN_1_IN: %MW342, H_CLOSE_1_IN: %MW344, M_CLOSE_1_IN: %MW346, H_OPEN_2_IN: %MW348, M_OPEN_2_IN: %MW350, H_CLOSE_2_IN: %MW352, M_CLOSE_2_IN: %MW354, H_OPEN_3_IN: %MW356, M_OPEN_3_IN: %MW358, H_CLOSE_3_IN: %MW360, M_CLOSE_3_IN: %MW362, KZH_OUT => %MX301.6) => %MX301.5
		EN --- LIMIT(60, %MW408, 9999) => %MW408
NETWORK 29
	*
		EN --- BB:BB(JZ_IN: %MX202.5, ZQ_IN: %MW408, BJ_IN: %MX202.0) => %MX203.0
_END_LD_
(* the same logic as Structured Text *)
(* Network 1: see the listing above *)
(* Network 2: see the listing above *)
(* Network 3 *)
T_R(CLK := TRUE);
T_DIAN := T_R.Q;
(* Network 4: see the listing above *)
(* Network 5: see the listing above *)
(* Network 6 *)
TD_TON(IN := TRUE, PT := T#10S);
ET := TD_TON.ET;
TD_TON_Q := TD_TON.Q;
(* Network 7: see the listing above *)
(* Network 8: see the listing above *)
(* Network 9: see the listing above *)
(* Network 10 *)
%MX202.6 := (%IX2.5 OR %MX300.7) AND (NOT %MX301.5 OR %MX301.6);
(* Network 11: see the listing above *)
(* Network 12: see the listing above *)
(* Network 13 *)
%MW302 := LIMIT(10, %MW302, 90);
(* Network 14: see the listing above *)
(* Network 15: see the listing above *)
(* Network 16: see the listing above *)
(* Network 17: see the listing above *)
(* Network 18: see the listing above *)
(* Network 19 *)
%QX2.5 := %QX2.4 AND (%MX211.6 AND %MX221.6 OR %MX211.6 AND %MX231.6 OR %MX221.6 AND %MX231.6);
(* Network 20 *)
%MW306 := LIMIT(2, %MW306, 9999);
%MW308 := LIMIT(2, %MW308, 9999);
(* Network 21 *)
FAN1(RJ_IN := %IX2.1, IN := FAN_1_KA, PSH_IN := PSH_Q_YSJ);
%QX2.6 := FAN1.OUT;
%MW870 := FAN1.ZHT_ROM;
%MX201.1 := FAN1.BJ_OUT;
FAN2(RJ_IN := %IX2.2, IN := FAN_2_KA, PSH_IN := PSH_Q_YSJ);
%QX2.7 := FAN2.OUT;
%MW872 := FAN2.ZHT_ROM;
%MX201.2 := FAN2.BJ_OUT;
SHB(RJ_IN := %IX2.3, IN := SHB_KA, PSH_IN := PSH_Q_YSJ);
%QX4.0 := SHB.OUT;
%MW878 := SHB.ZHT_ROM;
%MX201.5 := SHB.BJ_OUT;
(* Network 22: see the listing above *)
(* Network 23: see the listing above *)
(* Network 24 *)
(*机组报警*)%MX202.0 := ((*1#压缩机报警*)%MX210.0) AND NOT ((*1#卸载输出*)%MX300.1) OR ((*2#压缩机报警*)%MX220.0) AND NOT ((*2#卸载输出*)%MX300.2) OR ((*3#压缩机报警*)%MX230.0) AND NOT ((*3#卸载输出*)%MX300.3) OR %MX240.0 AND NOT %MX300.4 OR %MX250.0 AND NOT %MX300.5 OR ((*蒸发冷风扇2报警*)%MX200.0) OR %MX200.2 OR %MX200.3 OR %MX200.4 OR %MX200.5 OR %MX200.6 OR ((*油位报警*)%MX200.7) OR %MX201.1 OR ((*锁*)%MX201.2) OR ((*排气低温报警*)%MX201.3) OR ((*排气高温报警*)%MX201.4) OR ((*急停输出*)%MX201.5) OR %MX201.6 OR %MX201.7 OR ROOM1_ALA OR ROOM2_ALA OR ROOM3_ALA OR ROOM4_ALA OR ROOM5_ALA OR ROOM6_ALA OR ROOM7_ALA OR ROOM8_ALA OR ROOM9_ALA OR ROOM10_ALA OR ROOM11_ALA OR ROOM12_ALA OR %MX201.0 OR %MX583.6 OR %MX583.7 OR %MX203.1 OR %MX203.3 OR %MX1070.6 OR %MX1070.7;
%QX4.1 := (*机组报警*)%MX202.0;
(* Network 25: see the listing above *)
(* Network 26 *)
%MW482 := LIMIT(2, %MW482, 9999);
%MW484 := LIMIT(2, %MW484, 9999);
%MW486 := LIMIT(2, %MW486, 9999);
(* Network 27 *)
XH_YSH_1(WBKZL_IN := WBKZH, OPEN_IN := %MX202.6, DY_IN := %MW2000, MNL_XZH := XUZH_IN_1, MNL_HIGH_IN := SEL(%MX301.7, HIGH_IN_1, HIGH_IN_2), MNL_LOW_IN := SEL(%MX301.7, LOW_IN_1, LOW_IN_2), OPEN_YSH := %MW482, CLOSE_YSH := %MW484, JQ_OPEN_YSH := %MW486, JQ_1_BH_IN := CHD_1, JQ_2_BH_IN := CHD_2, JQ_3_BH_IN := CHD_3, JQ_4_BH_IN := CHT, JQ_5_BH_IN := CHT, JQ_6_BH_IN := CHT, DY_MU := 120, DY_MD := -10, JQ_NJ_SHU := JZ_NJ_SHU_1, WD_IN := %MW2016, XQ_WD_XZH := XQ_WD_XZH, WD_MU := 500, WD_MD := -500, GRD_IN := %MW472, GRD_YSH_SET := %MW474, TD_R := TD_TON_Q, TJ_ZHH := %MX301.2, YSJ_IN := %MX202.5, RESET := %MX202.7);
BH_WD := XH_YSH_1.YL_T_OUT;
%MW866 := XH_YSH_1.XH_T_XSH;
%MW848 := XH_YSH_1.XH_SHU_OUT;
%MW868 := XH_YSH_1.XH_ZHT;
JJQ_DCF_1 := XH_YSH_1.JJQ_OUT;
XQ_1_T := XH_YSH_1.XQ_WD_OUT;
GRD_1_OUT := XH_YSH_1.GRD_OUT;
%MX200.2 := XH_YSH_1.GRD_ALA;
%MW846 := XH_YSH_1.GRD_YSH_XSH;
%MX301.3 := XH_YSH_1.TJ_ZHH_OUT;
YALI_OUT_1 := XH_YSH_1.MNL_OUT;
XH_NJ_1(JQ_1_NJ := %MW814, JQ_2_NJ := %MW824, JQ_3_NJ := %MW834, JQ_4_NJ := %MW844, JQ_5_NJ := %MW854, JQ_6_NJ := %MW864, JQ_1_IN := %MX211.6, JQ_2_IN := %MX221.6, JQ_3_IN := %MX231.6, JQ_4_IN := %MX241.6, JQ_5_IN := %MX251.6, JQ_6_IN := %MX261.6);
JZ_NJ_SHU_1 := XH_NJ_1.JQ_NJ_ROM;
(* Network 28: see the listing above *)
(* Network 29 *)
BB(JZ_IN := %MX202.5, ZQ_IN := %MW408, BJ_IN := %MX202.0);
%MX203.0 := BB.CF_OUT;
END_PROGRAM

(* POU JIQI_KONGZHI, LD *)
  FUNCTION_BLOCK JIQI_KONGZHI
VAR_INPUT
	ON_OFF: BOOL;
	T_DIAN: BOOL;
	OPEN_ONE_IN: BOOL;
	OPEN_TWO_IN: BOOL;
	OPEN_THREE_IN: BOOL;
	SHD_IN: BOOL;
       BAOHU: BOOL;
	CLOSE_TIME: WORD;
	PSH_IN: BOOL;
	XIEZAI: BOOL;
	SUO_IN: BOOL;
	HIGHT_IN: BOOL;
	KU_KA: BOOL;
	WBKZ: BOOL;
	JJQ: BOOL;
	JZ_IN: BOOL;
END_VAR
VAR_OUTPUT
	OUT_ONE: BOOL;
	OUT_TWO: BOOL;
	OUT_25: BOOL;
	OUT_50: BOOL;
	OUT_75: BOOL;
	JJQ_OUT: BOOL;
	DCF_OUT: BOOL;
	ZHUANGTAI_OUT: BOOL;
	ET_OUT: WORD;
	SHUZI: WORD;
	OUT_KA: BOOL;
	JJQ_KA: BOOL;
	DCF_KA: BOOL;
END_VAR
VAR
	T_YASHI: TON;
	BAOJING_OUT: BOOL;
	OUT_100: BOOL;
	ET_TON_YASHI: TIME;
	T_YASHI_Q: BOOL;
	CLOSE: YANSHI_CLOSE;
	TOF_25: TOF;
	ET_TOF_25: TIME;
	T_25: TON;
	ET_T_25: TIME;
	T_50: TON;
	ET_T_50: TIME;
	T_75: TON;
	ET_T_75: TIME;
	OUT_50_KA: BOOL;
	OUT_75_KA: BOOL;
	SHD_KA: BOOL;
	BLINK: BLINK;
	KA_OFF: BOOL;
	R_TRIG: R_TRIG;
	JSHU: WORD;
	R_QL: R_TRIG;
END_VAR
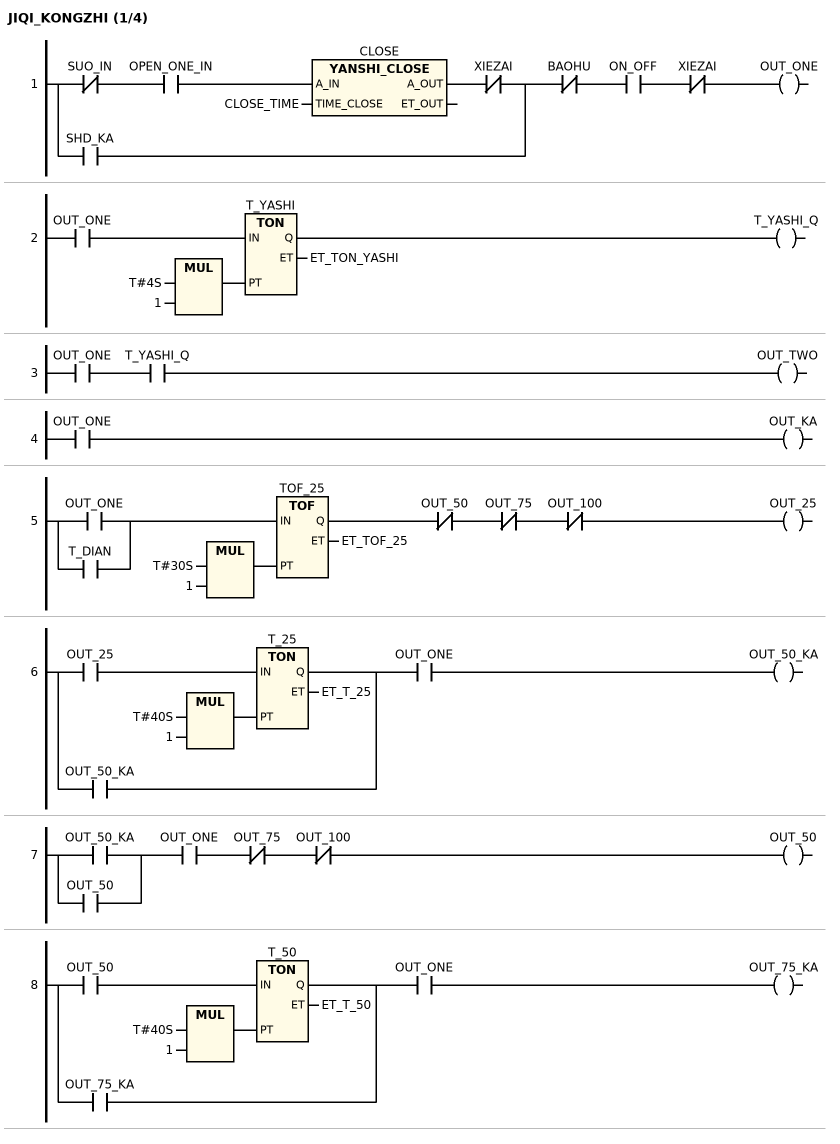
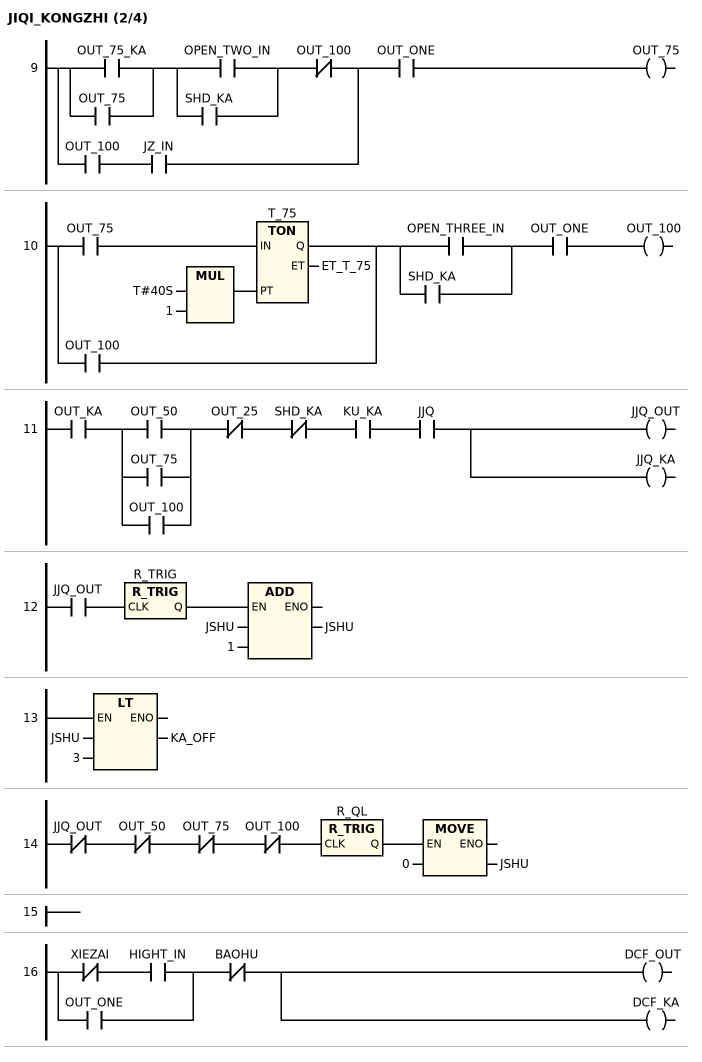
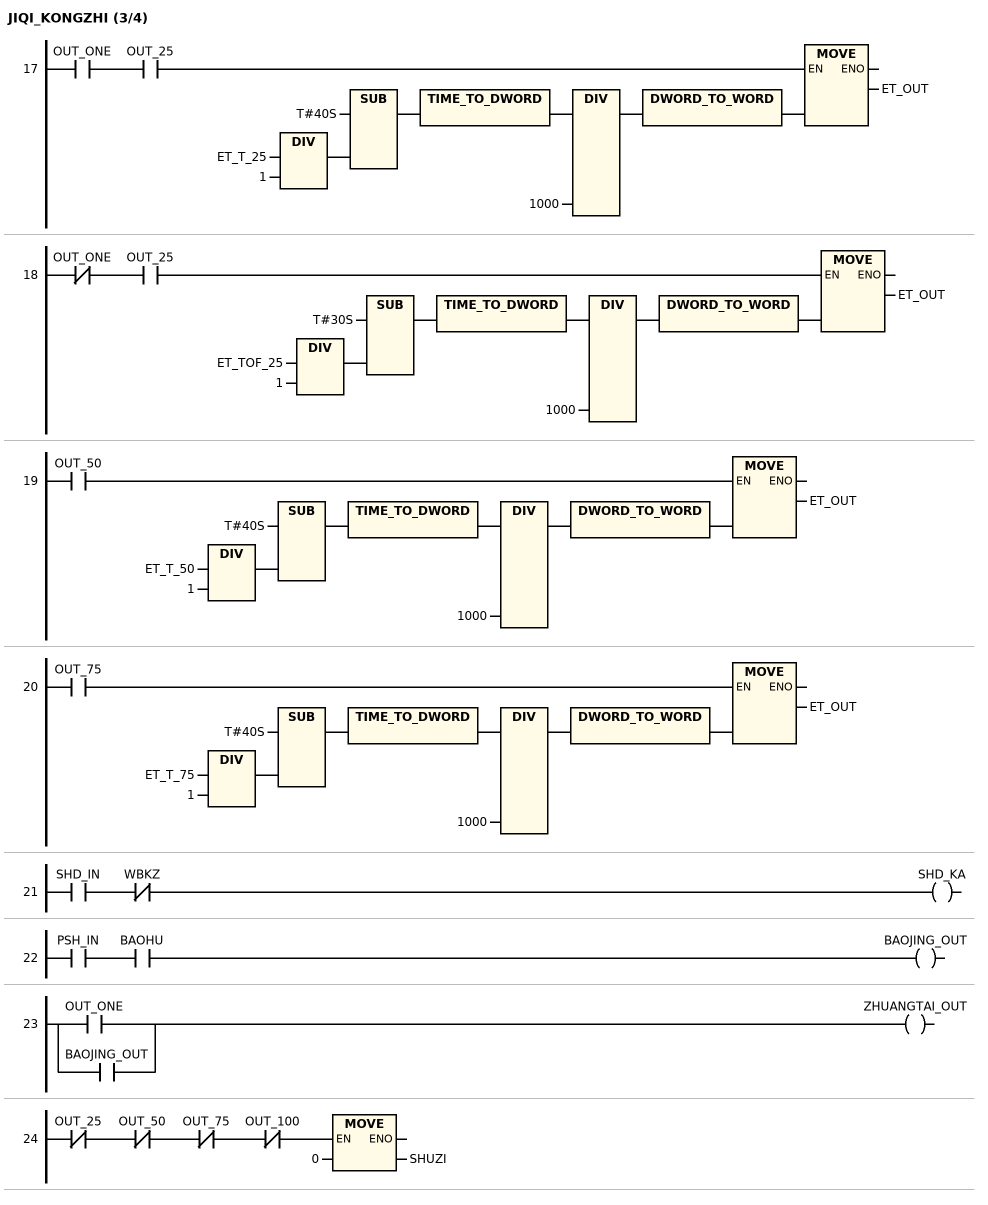
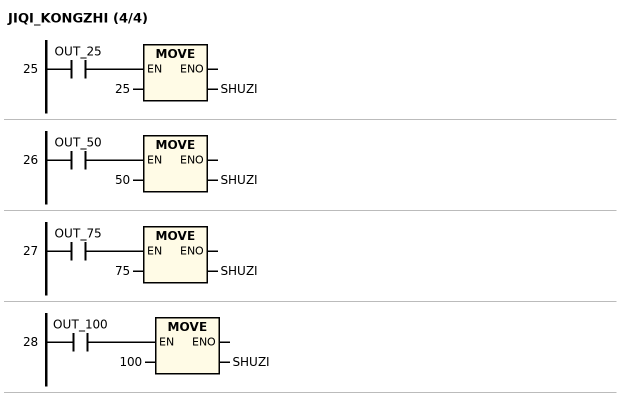
_LD_ (* Ladder Diagram *)
NETWORK 1
	{ [/SUO_IN] - [OPEN_ONE_IN] - CLOSE:YANSHI_CLOSE(A_IN: *, TIME_CLOSE: CLOSE_TIME) - [/XIEZAI] | [SHD_KA] } - [/BAOHU] - [ON_OFF] - [/XIEZAI] --- (OUT_ONE)
NETWORK 2
	[OUT_ONE] - T_YASHI:TON(IN: *, PT: MUL(T#4S, 1), ET => ET_TON_YASHI) --- (T_YASHI_Q)
NETWORK 3
	[OUT_ONE] - [T_YASHI_Q] --- (OUT_TWO)
NETWORK 4
	[OUT_ONE] --- (OUT_KA)
NETWORK 5
	{ [OUT_ONE] | [T_DIAN] } - TOF_25:TOF(IN: *, PT: MUL(T#30S, 1), ET => ET_TOF_25) - [/OUT_50] - [/OUT_75] - [/OUT_100] --- (OUT_25)
NETWORK 6
	{ [OUT_25] - T_25:TON(IN: *, PT: MUL(T#40S, 1), ET => ET_T_25) | [OUT_50_KA] } - [OUT_ONE] --- (OUT_50_KA)
NETWORK 7
	{ [OUT_50_KA] | [OUT_50] } - [OUT_ONE] - [/OUT_75] - [/OUT_100] --- (OUT_50)
NETWORK 8
	{ [OUT_50] - T_50:TON(IN: *, PT: MUL(T#40S, 1), ET => ET_T_50) | [OUT_75_KA] } - [OUT_ONE] --- (OUT_75_KA)
NETWORK 9
	{ { [OUT_75_KA] | [OUT_75] } - { [OPEN_TWO_IN] | [SHD_KA] } - [/OUT_100] | [OUT_100] - [JZ_IN] } - [OUT_ONE] --- (OUT_75)
NETWORK 10
	{ [OUT_75] - T_75:TON(IN: *, PT: MUL(T#40S, 1), ET => ET_T_75) | [OUT_100] } - { [OPEN_THREE_IN] | [SHD_KA] } - [OUT_ONE] --- (OUT_100)
NETWORK 11
	[OUT_KA] - { [OUT_50] | [OUT_75] | [OUT_100] } - [/OUT_25] - [/SHD_KA] - [KU_KA] - [JJQ] --- (JJQ_OUT) (JJQ_KA)
NETWORK 12
	[JJQ_OUT] - R_TRIG:R_TRIG(CLK: *)
		EN --- ADD(JSHU, 1) => JSHU
NETWORK 13
	*
		EN --- LT(JSHU, 3) => KA_OFF
NETWORK 14
	[/JJQ_OUT] - [/OUT_50] - [/OUT_75] - [/OUT_100] - R_QL:R_TRIG(CLK: *)
		EN --- MOVE(0) => JSHU
NETWORK 15
	*
NETWORK 16
	{ [/XIEZAI] - [HIGHT_IN] | [OUT_ONE] } - [/BAOHU] --- (DCF_OUT) (DCF_KA)
NETWORK 17
	[OUT_ONE] - [OUT_25]
		EN --- MOVE(DWORD_TO_WORD(DIV(TIME_TO_DWORD(SUB(T#40S, DIV(ET_T_25, 1))), 1000))) => ET_OUT
NETWORK 18
	[/OUT_ONE] - [OUT_25]
		EN --- MOVE(DWORD_TO_WORD(DIV(TIME_TO_DWORD(SUB(T#30S, DIV(ET_TOF_25, 1))), 1000))) => ET_OUT
NETWORK 19
	[OUT_50]
		EN --- MOVE(DWORD_TO_WORD(DIV(TIME_TO_DWORD(SUB(T#40S, DIV(ET_T_50, 1))), 1000))) => ET_OUT
NETWORK 20
	[OUT_75]
		EN --- MOVE(DWORD_TO_WORD(DIV(TIME_TO_DWORD(SUB(T#40S, DIV(ET_T_75, 1))), 1000))) => ET_OUT
NETWORK 21
	[SHD_IN] - [/WBKZ] --- (SHD_KA)
NETWORK 22
	[PSH_IN] - [BAOHU] --- (BAOJING_OUT)
NETWORK 23
	{ [OUT_ONE] | [BAOJING_OUT] } --- (ZHUANGTAI_OUT)
NETWORK 24
	[/OUT_25] - [/OUT_50] - [/OUT_75] - [/OUT_100]
		EN --- MOVE(0) => SHUZI
NETWORK 25
	[OUT_25]
		EN --- MOVE(25) => SHUZI
NETWORK 26
	[OUT_50]
		EN --- MOVE(50) => SHUZI
NETWORK 27
	[OUT_75]
		EN --- MOVE(75) => SHUZI
NETWORK 28
	[OUT_100]
		EN --- MOVE(100) => SHUZI
_END_LD_
(* the same logic as Structured Text *)
(* Network 1 *)
CLOSE(A_IN := NOT SUO_IN AND OPEN_ONE_IN, TIME_CLOSE := CLOSE_TIME);
OUT_ONE := (CLOSE.A_OUT AND NOT XIEZAI OR SHD_KA) AND NOT BAOHU AND ON_OFF AND NOT XIEZAI;
(* Network 2 *)
T_YASHI(IN := OUT_ONE, PT := T#4S * 1);
ET_TON_YASHI := T_YASHI.ET;
T_YASHI_Q := T_YASHI.Q;
(* Network 3 *)
OUT_TWO := OUT_ONE AND T_YASHI_Q;
(* Network 4 *)
OUT_KA := OUT_ONE;
(* Network 5 *)
TOF_25(IN := OUT_ONE OR T_DIAN, PT := T#30S * 1);
ET_TOF_25 := TOF_25.ET;
OUT_25 := TOF_25.Q AND NOT OUT_50 AND NOT OUT_75 AND NOT OUT_100;
(* Network 6 *)
T_25(IN := OUT_25, PT := T#40S * 1);
ET_T_25 := T_25.ET;
OUT_50_KA := (T_25.Q OR OUT_50_KA) AND OUT_ONE;
(* Network 7 *)
OUT_50 := (OUT_50_KA OR OUT_50) AND OUT_ONE AND NOT OUT_75 AND NOT OUT_100;
(* Network 8 *)
T_50(IN := OUT_50, PT := T#40S * 1);
ET_T_50 := T_50.ET;
OUT_75_KA := (T_50.Q OR OUT_75_KA) AND OUT_ONE;
(* Network 9 *)
OUT_75 := ((OUT_75_KA OR OUT_75) AND (OPEN_TWO_IN OR SHD_KA) AND NOT OUT_100 OR OUT_100 AND JZ_IN) AND OUT_ONE;
(* Network 10 *)
T_75(IN := OUT_75, PT := T#40S * 1);
ET_T_75 := T_75.ET;
OUT_100 := (T_75.Q OR OUT_100) AND (OPEN_THREE_IN OR SHD_KA) AND OUT_ONE;
(* Network 11 *)
JJQ_OUT := OUT_KA AND (OUT_50 OR OUT_75 OR OUT_100) AND NOT OUT_25 AND NOT SHD_KA AND KU_KA AND JJQ;
JJQ_KA := JJQ_OUT;
(* Network 12 *)
R_TRIG(CLK := JJQ_OUT);
IF R_TRIG.Q THEN
	JSHU := JSHU + 1;
END_IF;
(* Network 13 *)
KA_OFF := JSHU < 3;
(* Network 14 *)
R_QL(CLK := NOT JJQ_OUT AND NOT OUT_50 AND NOT OUT_75 AND NOT OUT_100);
IF R_QL.Q THEN
	JSHU := 0;
END_IF;
(* Network 15 *)
(* Network 16 *)
DCF_OUT := (NOT XIEZAI AND HIGHT_IN OR OUT_ONE) AND NOT BAOHU;
DCF_KA := DCF_OUT;
(* Network 17 *)
IF OUT_ONE AND OUT_25 THEN
	ET_OUT := DWORD_TO_WORD(TIME_TO_DWORD(T#40S - (ET_T_25 / 1)) / 1000);
END_IF;
(* Network 18 *)
IF NOT OUT_ONE AND OUT_25 THEN
	ET_OUT := DWORD_TO_WORD(TIME_TO_DWORD(T#30S - (ET_TOF_25 / 1)) / 1000);
END_IF;
(* Network 19 *)
IF OUT_50 THEN
	ET_OUT := DWORD_TO_WORD(TIME_TO_DWORD(T#40S - (ET_T_50 / 1)) / 1000);
END_IF;
(* Network 20 *)
IF OUT_75 THEN
	ET_OUT := DWORD_TO_WORD(TIME_TO_DWORD(T#40S - (ET_T_75 / 1)) / 1000);
END_IF;
(* Network 21 *)
SHD_KA := SHD_IN AND NOT WBKZ;
(* Network 22 *)
BAOJING_OUT := PSH_IN AND BAOHU;
(* Network 23 *)
ZHUANGTAI_OUT := OUT_ONE OR BAOJING_OUT;
(* Network 24 *)
IF NOT OUT_25 AND NOT OUT_50 AND NOT OUT_75 AND NOT OUT_100 THEN
	SHUZI := 0;
END_IF;
(* Network 25 *)
IF OUT_25 THEN
	SHUZI := 25;
END_IF;
(* Network 26 *)
IF OUT_50 THEN
	SHUZI := 50;
END_IF;
(* Network 27 *)
IF OUT_75 THEN
	SHUZI := 75;
END_IF;
(* Network 28 *)
IF OUT_100 THEN
	SHUZI := 100;
END_IF;
END_FUNCTION_BLOCK

(* POU YANSHI_CLOSE, LD *)
FUNCTION_BLOCK YANSHI_CLOSE
VAR_INPUT
	A_IN: BOOL;
END_VAR
VAR_OUTPUT
	A_OUT: BOOL;
	ET_OUT: WORD;
END_VAR
VAR
	TOF_A_OUT: BOOL;
	TOF_A: TOF;
	TOF_PT: TIME;
	TOF_ET: TIME;
	ET_KA: WORD;
END_VAR

VAR_INPUT RETAIN
	TIME_CLOSE: WORD;
END_VAR
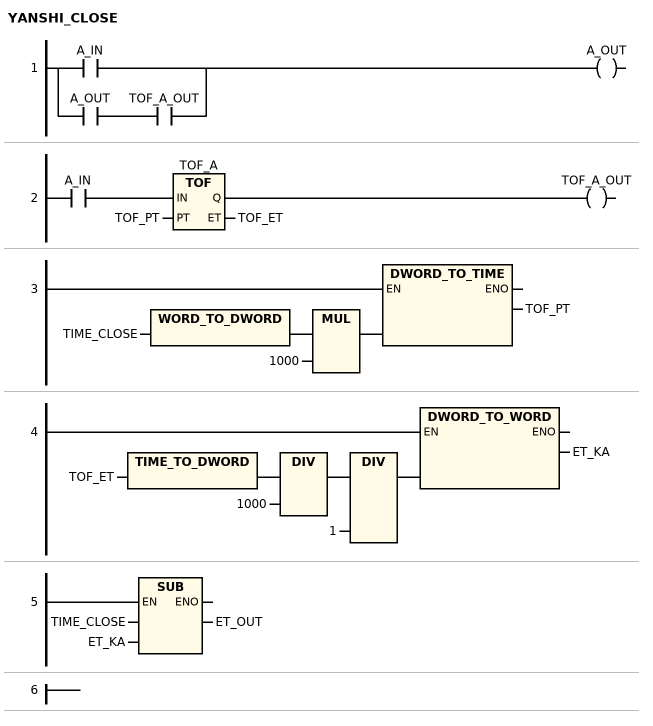
_LD_ (* Ladder Diagram *)
NETWORK 1
	{ [A_IN] | [A_OUT] - [TOF_A_OUT] } --- (A_OUT)
NETWORK 2
	[A_IN] - TOF_A:TOF(IN: *, PT: TOF_PT, ET => TOF_ET) --- (TOF_A_OUT)
NETWORK 3
	*
		EN --- DWORD_TO_TIME(MUL(WORD_TO_DWORD(TIME_CLOSE), 1000)) => TOF_PT
NETWORK 4
	*
		EN --- DWORD_TO_WORD(DIV(DIV(TIME_TO_DWORD(TOF_ET), 1000), 1)) => ET_KA
NETWORK 5
	*
		EN --- SUB(TIME_CLOSE, ET_KA) => ET_OUT
NETWORK 6
	*
_END_LD_
(* the same logic as Structured Text *)
(* Network 1 *)
A_OUT := A_IN OR A_OUT AND TOF_A_OUT;
(* Network 2 *)
TOF_A(IN := A_IN, PT := TOF_PT);
TOF_ET := TOF_A.ET;
TOF_A_OUT := TOF_A.Q;
(* Network 3 *)
TOF_PT := DWORD_TO_TIME(WORD_TO_DWORD(TIME_CLOSE) * 1000);
(* Network 4 *)
ET_KA := DWORD_TO_WORD((TIME_TO_DWORD(TOF_ET) / 1000) / 1);
(* Network 5 *)
ET_OUT := TIME_CLOSE - ET_KA;
(* Network 6 *)
END_FUNCTION_BLOCK

(* POU ZJSHQ, LD *)
  FUNCTION_BLOCK ZJSHQ
VAR_INPUT
	JIQI1_RST: BOOL;
	JIQI1: BOOL;
	JIQI2_RST: BOOL;
	JIQI2: BOOL;
	JIQI3_RST: BOOL;
	JIQI3: BOOL;
	JIQI4_RST: BOOL;
	JIQI4: BOOL;
	JIQI5_RST: BOOL;
	JIQI5: BOOL;
	JIQI6_RST: BOOL;
	JIQI6: BOOL;

END_VAR
VAR_OUTPUT
	JIQI1_H: DWORD;
	JIQI1_M: WORD;
	JIQI1_S: WORD;
	JIQI2_H: DWORD;
	JIQI2_M: WORD;
	JIQI2_S: WORD;
	JIQI3_H: DWORD;
	JIQI3_M: WORD;
	JIQI3_S: WORD;
	JIQI4_H: DWORD;
	JIQI4_M: WORD;
	JIQI4_S: WORD;
	JIQI5_H: DWORD;
	JIQI5_M: WORD;
	JIQI5_S: WORD;
	JIQI6_H: DWORD;
	JIQI6_M: WORD;
	JIQI6_S: WORD;




END_VAR
VAR
	JISHIQI_1HAO: JSHQ;
	JISHIQI_2HAO:  JSHQ;
	JISHIQI_3HAO:  JSHQ;
	JISHIQI_4HAO:  JSHQ;
	JISHIQI_5HAO:  JSHQ;
	JISHIQI_6HAO: JSHQ;


END_VAR
VAR_IN_OUT

END_VAR
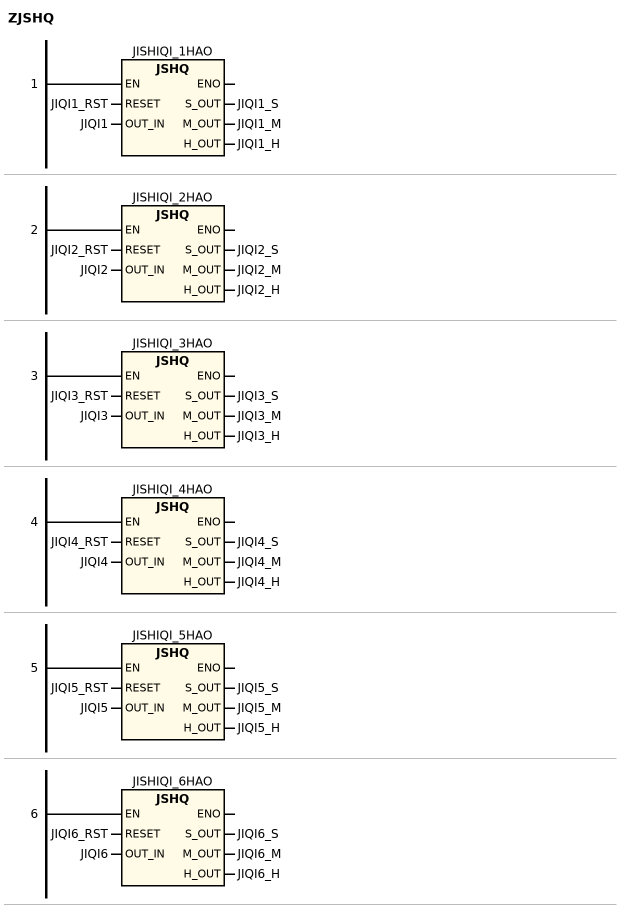
_LD_ (* Ladder Diagram *)
NETWORK 1
	*
		EN --- JISHIQI_1HAO:JSHQ(RESET: JIQI1_RST, OUT_IN: JIQI1, M_OUT => JIQI1_M, H_OUT => JIQI1_H) => JIQI1_S
NETWORK 2
	*
		EN --- JISHIQI_2HAO:JSHQ(RESET: JIQI2_RST, OUT_IN: JIQI2, M_OUT => JIQI2_M, H_OUT => JIQI2_H) => JIQI2_S
NETWORK 3
	*
		EN --- JISHIQI_3HAO:JSHQ(RESET: JIQI3_RST, OUT_IN: JIQI3, M_OUT => JIQI3_M, H_OUT => JIQI3_H) => JIQI3_S
NETWORK 4
	*
		EN --- JISHIQI_4HAO:JSHQ(RESET: JIQI4_RST, OUT_IN: JIQI4, M_OUT => JIQI4_M, H_OUT => JIQI4_H) => JIQI4_S
NETWORK 5
	*
		EN --- JISHIQI_5HAO:JSHQ(RESET: JIQI5_RST, OUT_IN: JIQI5, M_OUT => JIQI5_M, H_OUT => JIQI5_H) => JIQI5_S
NETWORK 6
	*
		EN --- JISHIQI_6HAO:JSHQ(RESET: JIQI6_RST, OUT_IN: JIQI6, M_OUT => JIQI6_M, H_OUT => JIQI6_H) => JIQI6_S
_END_LD_
(* the same logic as Structured Text *)
(* Network 1 *)
JISHIQI_1HAO(RESET := JIQI1_RST, OUT_IN := JIQI1);
JIQI1_M := JISHIQI_1HAO.M_OUT;
JIQI1_H := JISHIQI_1HAO.H_OUT;
JIQI1_S := JISHIQI_1HAO.S_OUT;
(* Network 2 *)
JISHIQI_2HAO(RESET := JIQI2_RST, OUT_IN := JIQI2);
JIQI2_M := JISHIQI_2HAO.M_OUT;
JIQI2_H := JISHIQI_2HAO.H_OUT;
JIQI2_S := JISHIQI_2HAO.S_OUT;
(* Network 3 *)
JISHIQI_3HAO(RESET := JIQI3_RST, OUT_IN := JIQI3);
JIQI3_M := JISHIQI_3HAO.M_OUT;
JIQI3_H := JISHIQI_3HAO.H_OUT;
JIQI3_S := JISHIQI_3HAO.S_OUT;
(* Network 4 *)
JISHIQI_4HAO(RESET := JIQI4_RST, OUT_IN := JIQI4);
JIQI4_M := JISHIQI_4HAO.M_OUT;
JIQI4_H := JISHIQI_4HAO.H_OUT;
JIQI4_S := JISHIQI_4HAO.S_OUT;
(* Network 5 *)
JISHIQI_5HAO(RESET := JIQI5_RST, OUT_IN := JIQI5);
JIQI5_M := JISHIQI_5HAO.M_OUT;
JIQI5_H := JISHIQI_5HAO.H_OUT;
JIQI5_S := JISHIQI_5HAO.S_OUT;
(* Network 6 *)
JISHIQI_6HAO(RESET := JIQI6_RST, OUT_IN := JIQI6);
JIQI6_M := JISHIQI_6HAO.M_OUT;
JIQI6_H := JISHIQI_6HAO.H_OUT;
JIQI6_S := JISHIQI_6HAO.S_OUT;
END_FUNCTION_BLOCK

(* POU JSHQ, LD *)
FUNCTION_BLOCK JSHQ
VAR_INPUT
	RESET: BOOL;
	OUT_IN: BOOL;
END_VAR
VAR_OUTPUT
	S_OUT: WORD;
	M_OUT: WORD;
	H_OUT: DWORD;
END_VAR
VAR
	TP_S: TP;
	 ET_OUT: TIME;
	CTU_M_OUT: BOOL;


	TP_S_OUT: BOOL;
	CTU_S_OUT: BOOL;
	R_H: R_TRIG;
END_VAR
VAR RETAIN
	CTU_M: CTU;
	CTU_S: CTU;
END_VAR
VAR_IN_OUT

END_VAR
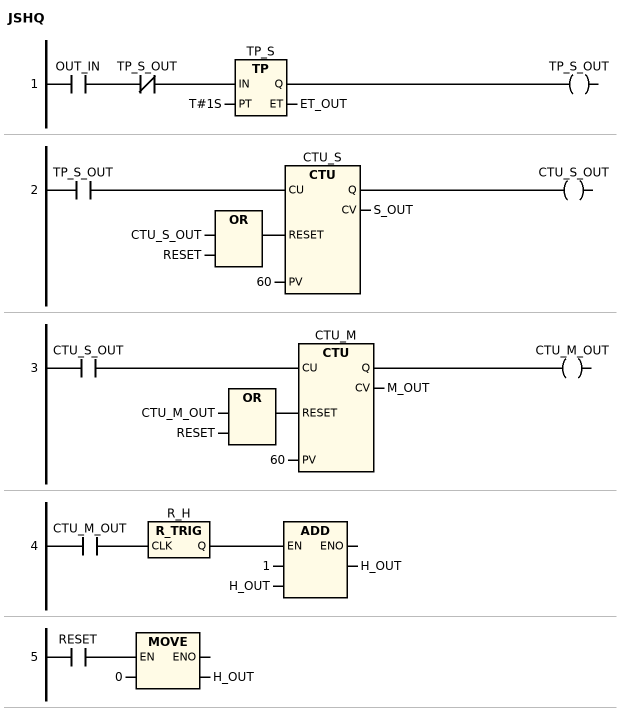
_LD_ (* Ladder Diagram *)
NETWORK 1
	[OUT_IN] - [/TP_S_OUT] - TP_S:TP(IN: *, PT: T#1S, ET => ET_OUT) --- (TP_S_OUT)
NETWORK 2
	[TP_S_OUT] - CTU_S:CTU(CU: *, RESET: OR(CTU_S_OUT, RESET), PV: 60, CV => S_OUT) --- (CTU_S_OUT)
NETWORK 3
	[CTU_S_OUT] - CTU_M:CTU(CU: *, RESET: OR(CTU_M_OUT, RESET), PV: 60, CV => M_OUT) --- (CTU_M_OUT)
NETWORK 4
	[CTU_M_OUT] - R_H:R_TRIG(CLK: *)
		EN --- ADD(1, H_OUT) => H_OUT
NETWORK 5
	[RESET]
		EN --- MOVE(0) => H_OUT
_END_LD_
(* the same logic as Structured Text *)
(* Network 1 *)
TP_S(IN := OUT_IN AND NOT TP_S_OUT, PT := T#1S);
ET_OUT := TP_S.ET;
TP_S_OUT := TP_S.Q;
(* Network 2 *)
CTU_S(CU := TP_S_OUT, RESET := CTU_S_OUT OR RESET, PV := 60);
S_OUT := CTU_S.CV;
CTU_S_OUT := CTU_S.Q;
(* Network 3 *)
CTU_M(CU := CTU_S_OUT, RESET := CTU_M_OUT OR RESET, PV := 60);
M_OUT := CTU_M.CV;
CTU_M_OUT := CTU_M.Q;
(* Network 4 *)
R_H(CLK := CTU_M_OUT);
IF R_H.Q THEN
	H_OUT := 1 + H_OUT;
END_IF;
(* Network 5 *)
IF RESET THEN
	H_OUT := 0;
END_IF;
END_FUNCTION_BLOCK

(* POU BAOHU_XIANSHI, LD *)
FUNCTION_BLOCK BAOHU_XIANSHI
VAR_INPUT
	ON_OFF: BOOL;
	REJIAN: BOOL;
	GAODIYA: BOOL;
	ZIBAO: BOOL;
	YOU_LL: BOOL;
	SHD_IN: BOOL;
	YOU_LV: BOOL;
	SHUCHU_1: BOOL;
	YOU_TIME_IN: WORD;
	XIE_ZAI: BOOL;
	RESET: BOOL;
	JG_YSH_SET: WORD;

END_VAR
VAR_OUTPUT
	BJ_OUT: BOOL;
	RJ_XH: BOOL;
	GDY_XH: BOOL;
	ZB_XH: BOOL;
	YOU_YA_XH: BOOL;
      YOU_LV_XH: BOOL;
	SHD_OUT: BOOL;
	ZHT_OUT: WORD;
	YOU_TIME_OUT: WORD;
	YSJ_CHD: BOOL;
	JG_YSH: WORD;
	CHD: BOOL;

END_VAR
VAR
	TON_YOU: TON;
	ET_TON_YOU: TIME;


	RJ_KA: BOOL;
	GDY_KA: BOOL;
	ZB_KA: BOOL;
	TON_OUT: BOOL;
	YOU_YA_KA: BOOL;
	SHD_TON: TON;
	SHD_R: R_TRIG;
	SHD_R_Q: BOOL;
	SHD_TON_Q: BOOL;
	DY_ZB_KA: BOOL;
	RJ_TON: TON;
	GDY_TOF: TOF;
	ZIBAO_TOF: TOF;
	DYZB_TOF: TOF;
	JG_OFF: BOOL;
	R_TRIG: R_TRIG;
	JG_CHD: BOOL;
	YANSHI_OPEN: YANSHI_OPEN;
	JG_ON: BOOL;
	YOU_LV_KA: BOOL;
	DYZB_Tn: TON;
END_VAR
VAR RETAIN
END_VAR
VAR_OUTPUT RETAIN

END_VAR
VAR_IN_OUT
END_VAR
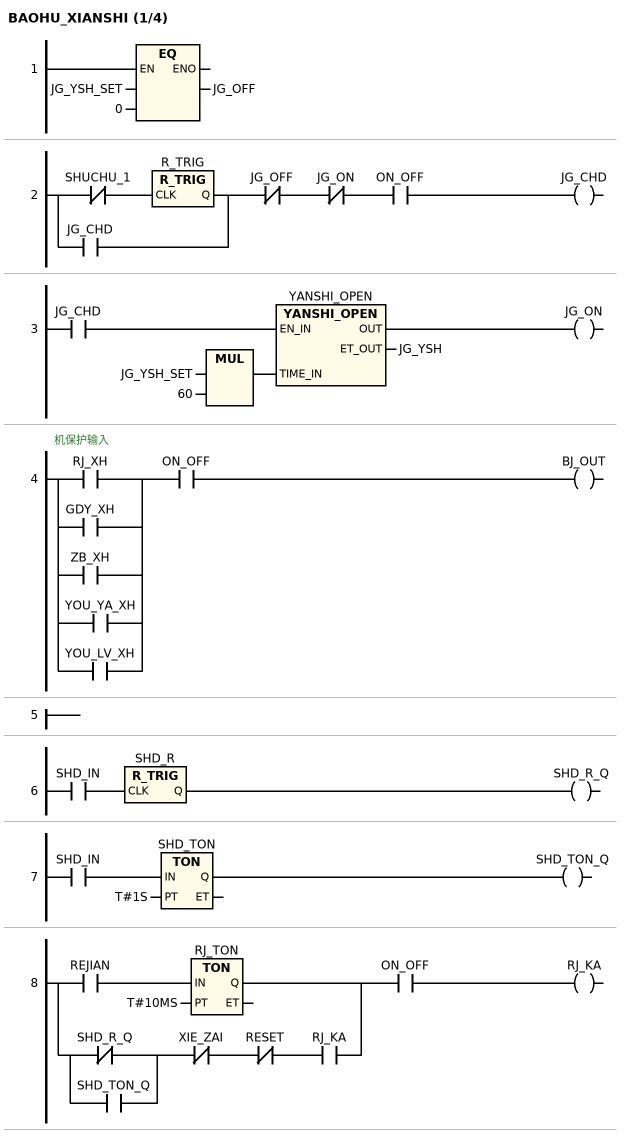
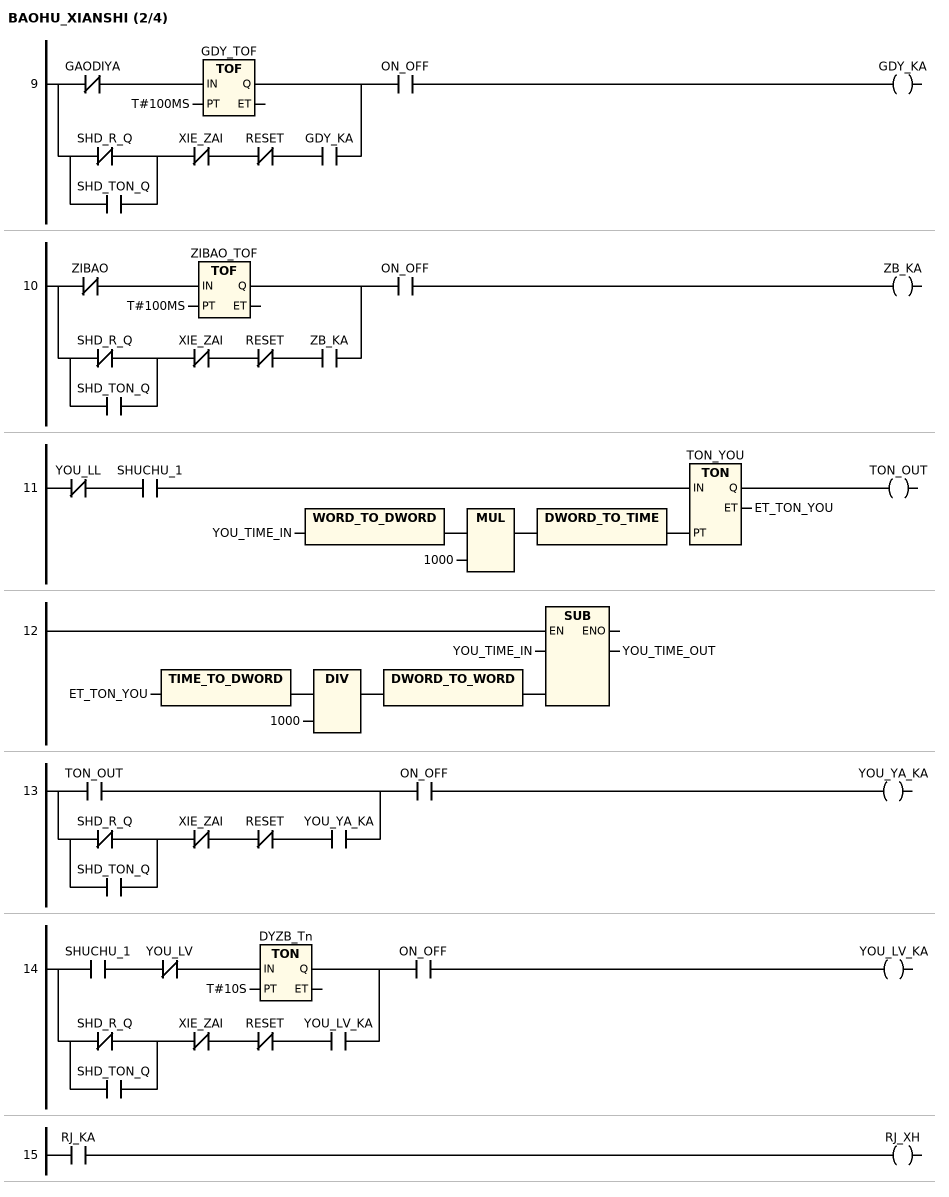
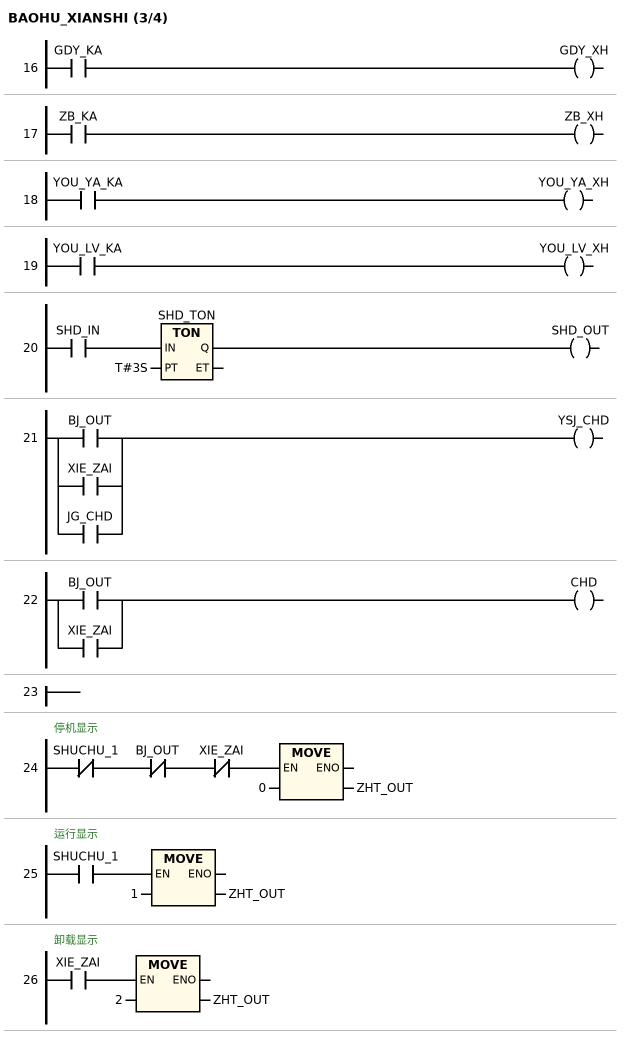
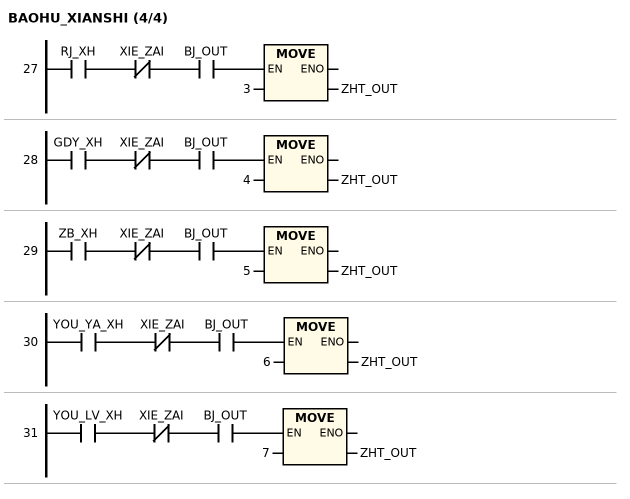
_LD_ (* Ladder Diagram *)
NETWORK 1
	*
		EN --- EQ(JG_YSH_SET, 0) => JG_OFF
NETWORK 2
	{ [/SHUCHU_1] - R_TRIG:R_TRIG(CLK: *) | [JG_CHD] } - [/JG_OFF] - [/JG_ON] - [ON_OFF] --- (JG_CHD)
NETWORK 3
	[JG_CHD] - YANSHI_OPEN:YANSHI_OPEN(EN_IN: *, TIME_IN: MUL(JG_YSH_SET, 60), ET_OUT => JG_YSH) --- (JG_ON)
NETWORK 4 (* 机保护输入 *)
	{ [RJ_XH] | [GDY_XH] | [ZB_XH] | [YOU_YA_XH] | [YOU_LV_XH] } - [ON_OFF] --- (BJ_OUT)
NETWORK 5
	*
NETWORK 6
	[SHD_IN] - SHD_R:R_TRIG(CLK: *) --- (SHD_R_Q)
NETWORK 7
	[SHD_IN] - SHD_TON:TON(IN: *, PT: T#1S) --- (SHD_TON_Q)
NETWORK 8
	{ [REJIAN] - RJ_TON:TON(IN: *, PT: T#10MS) | { [/SHD_R_Q] | [SHD_TON_Q] } - [/XIE_ZAI] - [/RESET] - [RJ_KA] } - [ON_OFF] --- (RJ_KA)
NETWORK 9
	{ [/GAODIYA] - GDY_TOF:TOF(IN: *, PT: T#100MS) | { [/SHD_R_Q] | [SHD_TON_Q] } - [/XIE_ZAI] - [/RESET] - [GDY_KA] } - [ON_OFF] --- (GDY_KA)
NETWORK 10
	{ [/ZIBAO] - ZIBAO_TOF:TOF(IN: *, PT: T#100MS) | { [/SHD_R_Q] | [SHD_TON_Q] } - [/XIE_ZAI] - [/RESET] - [ZB_KA] } - [ON_OFF] --- (ZB_KA)
NETWORK 11
	[/YOU_LL] - [SHUCHU_1] - TON_YOU:TON(IN: *, PT: DWORD_TO_TIME(MUL(WORD_TO_DWORD(YOU_TIME_IN), 1000)), ET => ET_TON_YOU) --- (TON_OUT)
NETWORK 12
	*
		EN --- SUB(YOU_TIME_IN, DWORD_TO_WORD(DIV(TIME_TO_DWORD(ET_TON_YOU), 1000))) => YOU_TIME_OUT
NETWORK 13
	{ [TON_OUT] | { [/SHD_R_Q] | [SHD_TON_Q] } - [/XIE_ZAI] - [/RESET] - [YOU_YA_KA] } - [ON_OFF] --- (YOU_YA_KA)
NETWORK 14
	{ [SHUCHU_1] - [/YOU_LV] - DYZB_Tn:TON(IN: *, PT: T#10S) | { [/SHD_R_Q] | [SHD_TON_Q] } - [/XIE_ZAI] - [/RESET] - [YOU_LV_KA] } - [ON_OFF] --- (YOU_LV_KA)
NETWORK 15
	[RJ_KA] --- (RJ_XH)
NETWORK 16
	[GDY_KA] --- (GDY_XH)
NETWORK 17
	[ZB_KA] --- (ZB_XH)
NETWORK 18
	[YOU_YA_KA] --- (YOU_YA_XH)
NETWORK 19
	[YOU_LV_KA] --- (YOU_LV_XH)
NETWORK 20
	[SHD_IN] - SHD_TON:TON(IN: *, PT: T#3S) --- (SHD_OUT)
NETWORK 21
	{ [BJ_OUT] | [XIE_ZAI] | [JG_CHD] } --- (YSJ_CHD)
NETWORK 22
	{ [BJ_OUT] | [XIE_ZAI] } --- (CHD)
NETWORK 23
	*
NETWORK 24 (* 停机显示 *)
	[/SHUCHU_1] - [/BJ_OUT] - [/XIE_ZAI]
		EN --- MOVE(0) => ZHT_OUT
NETWORK 25 (* 运行显示 *)
	[SHUCHU_1]
		EN --- MOVE(1) => ZHT_OUT
NETWORK 26 (* 卸载显示 *)
	[XIE_ZAI]
		EN --- MOVE(2) => ZHT_OUT
NETWORK 27
	[RJ_XH] - [/XIE_ZAI] - [BJ_OUT]
		EN --- MOVE(3) => ZHT_OUT
NETWORK 28
	[GDY_XH] - [/XIE_ZAI] - [BJ_OUT]
		EN --- MOVE(4) => ZHT_OUT
NETWORK 29
	[ZB_XH] - [/XIE_ZAI] - [BJ_OUT]
		EN --- MOVE(5) => ZHT_OUT
NETWORK 30
	[YOU_YA_XH] - [/XIE_ZAI] - [BJ_OUT]
		EN --- MOVE(6) => ZHT_OUT
NETWORK 31
	[YOU_LV_XH] - [/XIE_ZAI] - [BJ_OUT]
		EN --- MOVE(7) => ZHT_OUT
_END_LD_
(* the same logic as Structured Text *)
(* Network 1 *)
JG_OFF := JG_YSH_SET = 0;
(* Network 2 *)
R_TRIG(CLK := NOT SHUCHU_1);
JG_CHD := (R_TRIG.Q OR JG_CHD) AND NOT JG_OFF AND NOT JG_ON AND ON_OFF;
(* Network 3 *)
YANSHI_OPEN(EN_IN := JG_CHD, TIME_IN := JG_YSH_SET * 60);
JG_YSH := YANSHI_OPEN.ET_OUT;
JG_ON := YANSHI_OPEN.OUT;
(* Network 4: 机保护输入 *)
BJ_OUT := (RJ_XH OR GDY_XH OR ZB_XH OR YOU_YA_XH OR YOU_LV_XH) AND ON_OFF;
(* Network 5 *)
(* Network 6 *)
SHD_R(CLK := SHD_IN);
SHD_R_Q := SHD_R.Q;
(* Network 7 *)
SHD_TON(IN := SHD_IN, PT := T#1S);
SHD_TON_Q := SHD_TON.Q;
(* Network 8 *)
RJ_TON(IN := REJIAN, PT := T#10MS);
RJ_KA := (RJ_TON.Q OR (NOT SHD_R_Q OR SHD_TON_Q) AND NOT XIE_ZAI AND NOT RESET AND RJ_KA) AND ON_OFF;
(* Network 9 *)
GDY_TOF(IN := NOT GAODIYA, PT := T#100MS);
GDY_KA := (GDY_TOF.Q OR (NOT SHD_R_Q OR SHD_TON_Q) AND NOT XIE_ZAI AND NOT RESET AND GDY_KA) AND ON_OFF;
(* Network 10 *)
ZIBAO_TOF(IN := NOT ZIBAO, PT := T#100MS);
ZB_KA := (ZIBAO_TOF.Q OR (NOT SHD_R_Q OR SHD_TON_Q) AND NOT XIE_ZAI AND NOT RESET AND ZB_KA) AND ON_OFF;
(* Network 11 *)
TON_YOU(IN := NOT YOU_LL AND SHUCHU_1, PT := DWORD_TO_TIME(WORD_TO_DWORD(YOU_TIME_IN) * 1000));
ET_TON_YOU := TON_YOU.ET;
TON_OUT := TON_YOU.Q;
(* Network 12 *)
YOU_TIME_OUT := YOU_TIME_IN - DWORD_TO_WORD(TIME_TO_DWORD(ET_TON_YOU) / 1000);
(* Network 13 *)
YOU_YA_KA := (TON_OUT OR (NOT SHD_R_Q OR SHD_TON_Q) AND NOT XIE_ZAI AND NOT RESET AND YOU_YA_KA) AND ON_OFF;
(* Network 14 *)
DYZB_Tn(IN := SHUCHU_1 AND NOT YOU_LV, PT := T#10S);
YOU_LV_KA := (DYZB_Tn.Q OR (NOT SHD_R_Q OR SHD_TON_Q) AND NOT XIE_ZAI AND NOT RESET AND YOU_LV_KA) AND ON_OFF;
(* Network 15 *)
RJ_XH := RJ_KA;
(* Network 16 *)
GDY_XH := GDY_KA;
(* Network 17 *)
ZB_XH := ZB_KA;
(* Network 18 *)
YOU_YA_XH := YOU_YA_KA;
(* Network 19 *)
YOU_LV_XH := YOU_LV_KA;
(* Network 20 *)
SHD_TON(IN := SHD_IN, PT := T#3S);
SHD_OUT := SHD_TON.Q;
(* Network 21 *)
YSJ_CHD := BJ_OUT OR XIE_ZAI OR JG_CHD;
(* Network 22 *)
CHD := BJ_OUT OR XIE_ZAI;
(* Network 23 *)
(* Network 24: 停机显示 *)
IF NOT SHUCHU_1 AND NOT BJ_OUT AND NOT XIE_ZAI THEN
	ZHT_OUT := 0;
END_IF;
(* Network 25: 运行显示 *)
IF SHUCHU_1 THEN
	ZHT_OUT := 1;
END_IF;
(* Network 26: 卸载显示 *)
IF XIE_ZAI THEN
	ZHT_OUT := 2;
END_IF;
(* Network 27 *)
IF RJ_XH AND NOT XIE_ZAI AND BJ_OUT THEN
	ZHT_OUT := 3;
END_IF;
(* Network 28 *)
IF GDY_XH AND NOT XIE_ZAI AND BJ_OUT THEN
	ZHT_OUT := 4;
END_IF;
(* Network 29 *)
IF ZB_XH AND NOT XIE_ZAI AND BJ_OUT THEN
	ZHT_OUT := 5;
END_IF;
(* Network 30 *)
IF YOU_YA_XH AND NOT XIE_ZAI AND BJ_OUT THEN
	ZHT_OUT := 6;
END_IF;
(* Network 31 *)
IF YOU_LV_XH AND NOT XIE_ZAI AND BJ_OUT THEN
	ZHT_OUT := 7;
END_IF;
END_FUNCTION_BLOCK

(* POU YANSHI_OPEN, LD *)
FUNCTION_BLOCK YANSHI_OPEN
VAR_INPUT
	EN_IN: BOOL;
	TIME_IN: WORD;
END_VAR
VAR_OUTPUT
	OUT: BOOL;
	ET_OUT: WORD;
END_VAR
VAR
	T1: TON;
	PT: TIME;
	ET: TIME;
	ET_KA: WORD;
END_VAR
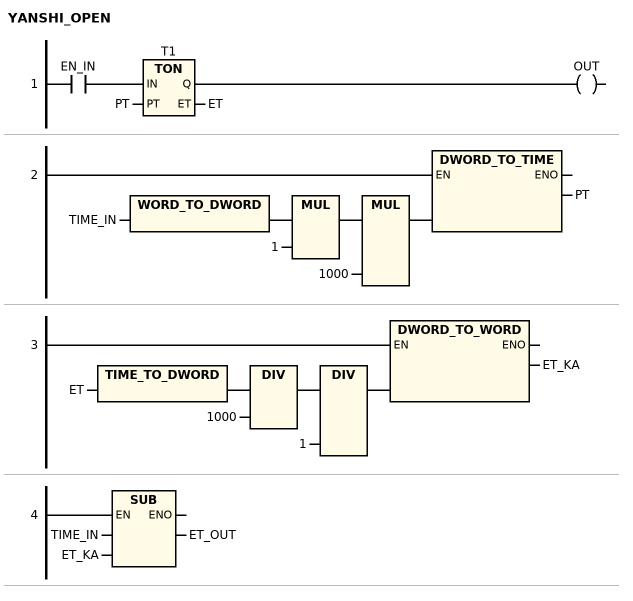
_LD_ (* Ladder Diagram *)
NETWORK 1
	[EN_IN] - T1:TON(IN: *, PT: PT, ET => ET) --- (OUT)
NETWORK 2
	*
		EN --- DWORD_TO_TIME(MUL(MUL(WORD_TO_DWORD(TIME_IN), 1), 1000)) => PT
NETWORK 3
	*
		EN --- DWORD_TO_WORD(DIV(DIV(TIME_TO_DWORD(ET), 1000), 1)) => ET_KA
NETWORK 4
	*
		EN --- SUB(TIME_IN, ET_KA) => ET_OUT
_END_LD_
(* the same logic as Structured Text *)
(* Network 1 *)
T1(IN := EN_IN, PT := PT);
ET := T1.ET;
OUT := T1.Q;
(* Network 2 *)
PT := DWORD_TO_TIME((WORD_TO_DWORD(TIME_IN) * 1) * 1000);
(* Network 3 *)
ET_KA := DWORD_TO_WORD((TIME_TO_DWORD(ET) / 1000) / 1);
(* Network 4 *)
ET_OUT := TIME_IN - ET_KA;
END_FUNCTION_BLOCK

(* POU BH_ZHFL, LD *)
FUNCTION_BLOCK BH_ZHFL
VAR_INPUT
	RJ_IN: BOOL;
	IN: BOOL;
	PSH_IN: BOOL;
END_VAR
VAR_OUTPUT
	BJ_OUT: BOOL;
	OUT: BOOL;
	OUT_KA: BOOL;
	OUT_ZHSH: BOOL;
	ZHT_ROM: WORD;
END_VAR
VAR

END_VAR
VAR RETAIN
END_VAR
